NETWORK
TITLE = **** 7.2 - Submodules - Command **** Check Received
// Check Received Data
      AN    #SendAckCmd;  // Send AckCmd
      JC    SACK;
      L     #OldRecMsgNbr;  // MessageNumber (SeqNbr)
      OPN   #I_VDCommSendDB;
      T     %DBW8;
      L     #OldSubSystem;  // Subsystem
      T     %DBW6;
      L     1;  // MessageType
      T     %DBW4;
      L     10;  //LengthLength
      T     %DBW2;
      JU    PAPM;
SACK: NOP   0;

      AN    #SendNackCmd;  // Send NackCmd
      JC    SNAC;
      L     #OldRecMsgNbr;  // MessageNumber (SeqNbr)
      OPN   #I_VDCommSendDB;
      T     %DBW8;
      L     #OldSubSystem;  // Subsystem
      T     %DBW6;
      L     0;  // MessageType
      T     %DBW4;
      L     10;  //LengthLength
      T     %DBW2;
      JU    PAPM;
SNAC: NOP   0;

      A     #SendApplMsgCmd;  // Send Application Message
      AN    #SendActive;
      AN    #SendDone;
      JCN   PAPM;

// Number of bytes to copy***************************************************************************************************
//     L     #I_VDCommSendDBBuf   // SEND BUF        APa Fixa S7-1500
//     T     #SS_Out_Buf          // DB number to copy
//     OPN DB [ #SS_Out_Buf]      // APa Fixa S7-1500
//     OPN   #I_VDCommSendDBBuf

      L     #IO_VD.VDCommSendDBNr;
      L     0;
      ==I;
//     JCN   NSrS1
      OPN   #IO_VD.VDCommSendDB;
      L     DBNO;
      T     #OutBuf;
      OPN   #IO_VD.VDCommSendDB;
      LAR1  P##PointerSendBuf;
      L     %DBW2;  // Length
      T     LW [AR1, P#2.0];
      OPN   #IO_VD.VDCommSendDB;
      LAR1  P##PointerSend;
      L     %DBW2;
      T     LW [AR1, P#2.0];
      OPN   #IO_VD.VDCommSendDB;
      L     DBNO;
      T     #OutBuf;
//NSrS1: NOP 0

//      OPN   #I_VDCommSendBufStn2 APa Fixa S7-1500
//    L DBNO
//   L     #I_VDCommSendDBBuf
//    ==I
//    L DBNO
//     T     #SS_Out_Buf
//     JCN   NSrS2
//      OPN   #I_VDCommSendBufStn2
//    L     %DBW2                // Length
//    T     %LW22                // SEND BUF
//     T     %LW12                // SEND
//     L DBNO
//      T     #SS_Out_Buf
//NSrS2: NOP 0

//*****************************************************************************************************************************


// Pointer to the Receive DB (Pointer_SEND_Buf) APa Fixa S7-1500
// DB no DB no
//    L DBNO
//  T     #SS_Out_Buf
//   L     #I_VDCommSendDBBuf
      OPN   #IO_VD.VDCommSendDB;
      L     DBNO;
      T     #OutBuf;
      L     #OutBuf;
      LAR1  P##PointerSendBuf;
      L     #OutBuf;
      T     LW [AR1, P#4.0];
//      T     %LW24                // SEND BUF
      CALL  BLKMOV
      ( SRCBLK  := #PointerSendBuf,  // SEND Buffer
        RET_VAL := "NotUsedInt",
        DSTBLK  := #PointerSend  // SEND
      );  // Copy data from buffer DB to send DB

      L     #SendMsgNbr;
      L     1000;
      >=I;
      JCN   ZermMsgCnt;
      L     1;
      T     #SendMsgNbr;

ZermMsgCnt:OPN   #I_VDCommSendDB;
      L     #SendMsgNbr;
      A     #AD_TimeoutApplMsgMem;
      JC    noin;
      L     #SendMsgNbr;
      +     1;
noin: T     #SendMsgNbr;
      T     %DBW8;  // Messagenumber

      CLR;
      R     #AD_TimeoutApplMsgMem;

PAPM: OPN   #I_VDCommSendDB;
      L     %DBW2;
      T     #MsgLen;

      L     1;
      T     %DBB0;

      A     #NackIsLastSent;
      A     #SendAckCmd;
      JCN   ZeroMesag;
      L     0;
      T     %DBW4;
ZeroMesag:NOP   0;

      L     #SendMsgNbr;
      T     "NotUsedDInt";

NETWORK
TITLE = **** 7.2 - Submodules - Command **** Length to Send Pointers
// Length to Send Pointers / Check Received Data
      LAR1  P##PointerSend;
      L     #MsgLen;
      T     LW [AR1, P#2.0];


REGION Network 73: **** 7.2 - Submodules - Command **** Send Data VD
   // Send Data VD
   #_w1 := (#SendNackCmd OR #SendAckCmd OR #SendApplMsgCmd OR #SendKeepAliveCmd) AND NOT #HMIResetAndInit AND NOT #SendActive;
   IF "TRUE" THEN
       #TSendVD(REQ := #_w1,   // TSEND
                ID := #ConnectionSettings.ID,
                LEN := #MsgLen,
                DATA := #PointerSend,
                DONE => #TSEND.Done,
                BUSY => #TSEND.Busy,
                ERROR => #TSEND.Error,
                STATUS => #TSEND.Status);
   END_IF;
   IF #_w1 THEN #TSEND.Sending := TRUE; END_IF;
END_REGION

NETWORK
TITLE = **** 7.2 - Submodules - Command **** Send Data to VD
// Send data to VD (length is the length in the SEND_DB)
      L     #TSEND.Status;
      L     16#0000;
      ==I;
      =     #SendJobCompleted;  // Send job completed without error
      L     #TSEND.Status;
      L     16#7000;
      ==I;
      =     #SendInactive;  // No job processing active
      L     #TSEND.Status;
      L     16#7001;
      ==I;
      =     #SendStartOfProc;  // Start of job processing, data being sent
      L     #TSEND.Status;
      L     16#7002;
      ==I;
      =     #SendFollowOnCall;  // Follow-on call (REQ irrelevant ), job being processed



REGION Network 75: **** 7.2 - Submodules - Command **** Send Status
   // Send Status to memory
   IF #TSEND.Error THEN #TSEND.Status_Mem := #TSEND.Status; END_IF;
END_REGION

REGION Network 76: **** 7.2 - Submodules - Command **** Stop Send
   // Stop sending  Error,Done,Sending AND NOT Busy
   IF (#TSEND.Sending AND NOT #TSEND.Busy AND #AD_SendTimeOut) OR #TSEND.Error OR #TSEND.Done THEN
       #TSEND.Sending := FALSE;
   END_IF;
END_REGION

REGION Network 77: **** 7.2 - Submodules - Command **** Send Active
   // Send Active
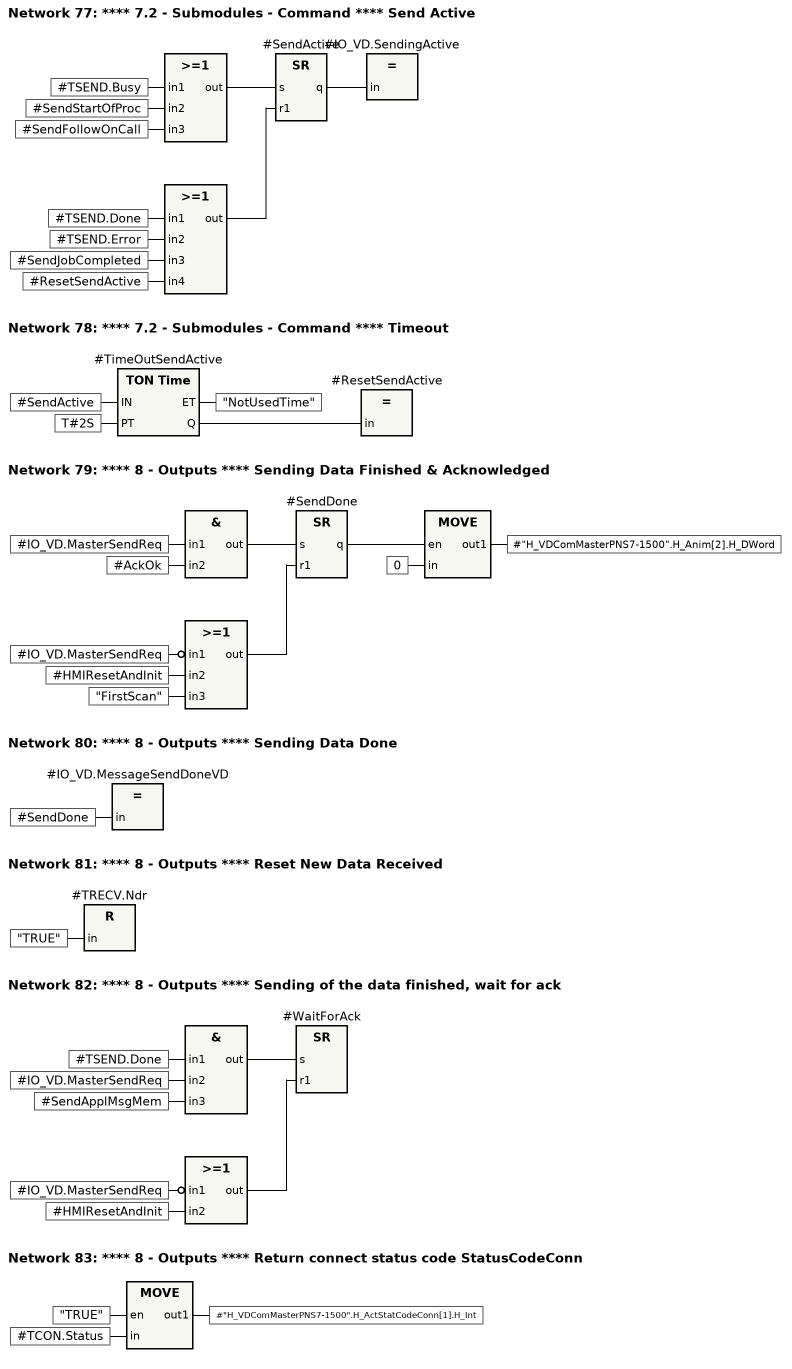
   IF #TSEND.Busy OR #SendStartOfProc OR #SendFollowOnCall THEN
       #SendActive := TRUE;   // SR flip-flop
   END_IF;
   IF #TSEND.Done OR #TSEND.Error OR #SendJobCompleted OR #ResetSendActive THEN #SendActive := FALSE; END_IF;
   #IO_VD.SendingActive := #SendActive;
END_REGION

REGION Network 78: **** 7.2 - Submodules - Command **** Timeout
   // Timeout
   #TimeOutSendActive(IN := #SendActive, PT := T#2S, ET => "NotUsedTime");   // TON
   #ResetSendActive := #TimeOutSendActive.Q;
END_REGION

REGION Network 79: **** 8 - Outputs **** Sending Data Finished & Acknowledged
   // Sending Data Finished & Acknowledged
   IF #IO_VD.MasterSendReq AND #AckOk THEN
       #SendDone := TRUE;   // SR flip-flop
   END_IF;
   IF NOT #IO_VD.MasterSendReq OR #HMIResetAndInit OR "FirstScan" THEN #SendDone := FALSE; END_IF;
   IF #SendDone THEN #"H_VDComMasterPNS7-1500".H_Anim[2].H_DWord := 0; END_IF;
END_REGION

REGION Network 80: **** 8 - Outputs **** Sending Data Done
   // Sending Data Done
   #IO_VD.MessageSendDoneVD := #SendDone;
END_REGION

REGION Network 81: **** 8 - Outputs **** Reset New Data Received
   // Reset "New data received" bit. All processing shall be done before this step.
   IF "TRUE" THEN #TRECV.Ndr := FALSE; END_IF;
END_REGION

REGION Network 82: **** 8 - Outputs **** Sending of the data finished, wait for ack
   // Sending of the data finished, wait for ack
   IF #TSEND.Done AND #IO_VD.MasterSendReq AND #SendApplMsgMem THEN
       #WaitForAck := TRUE;   // SR flip-flop
   END_IF;
   IF NOT #IO_VD.MasterSendReq OR #HMIResetAndInit THEN #WaitForAck := FALSE; END_IF;
END_REGION

REGION Network 83: **** 8 - Outputs **** Return connect status code StatusCodeConn
   // Return connect status code H_StatusCodeConn
   IF "TRUE" THEN #"H_VDComMasterPNS7-1500".H_ActStatCodeConn[1].H_Int := #TCON.Status; END_IF;
END_REGION

REGION Network 84: **** 8 - Outputs **** Return receive status code StatusCodeDisconn
   // Return receive status code H_StatusCodeDisconn
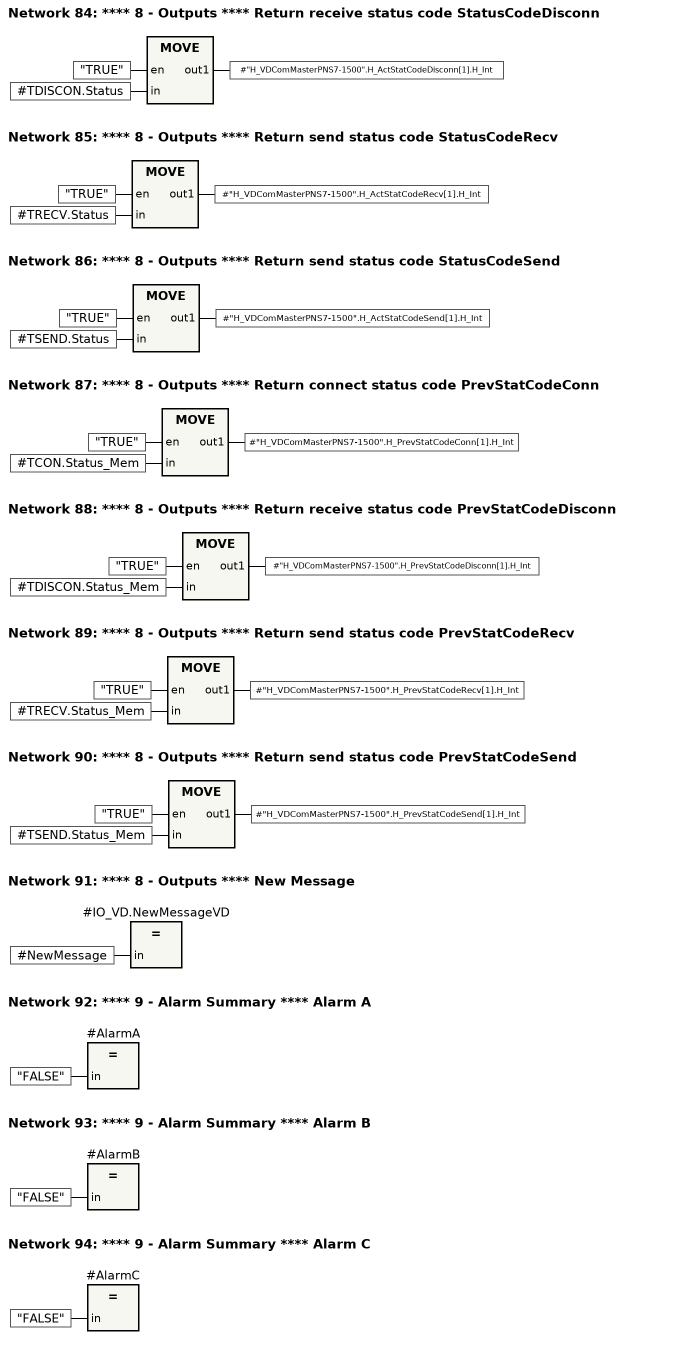
   IF "TRUE" THEN #"H_VDComMasterPNS7-1500".H_ActStatCodeDisconn[1].H_Int := #TDISCON.Status; END_IF;
END_REGION

REGION Network 85: **** 8 - Outputs **** Return send status code StatusCodeRecv
   // Return send status code H_StatusCodeRecv
   IF "TRUE" THEN #"H_VDComMasterPNS7-1500".H_ActStatCodeRecv[1].H_Int := #TRECV.Status; END_IF;
END_REGION

REGION Network 86: **** 8 - Outputs **** Return send status code StatusCodeSend
   // Return send status code H_StatusCodeSend
   IF "TRUE" THEN #"H_VDComMasterPNS7-1500".H_ActStatCodeSend[1].H_Int := #TSEND.Status; END_IF;
END_REGION

REGION Network 87: **** 8 - Outputs **** Return connect status code PrevStatCodeConn
   // Return connect status code H_PrevStatCodeConn
   IF "TRUE" THEN #"H_VDComMasterPNS7-1500".H_PrevStatCodeConn[1].H_Int := #TCON.Status_Mem; END_IF;
END_REGION

REGION Network 88: **** 8 - Outputs **** Return receive status code PrevStatCodeDisconn
   // Return receive status code H_PrevStatCodeDisconn
   IF "TRUE" THEN #"H_VDComMasterPNS7-1500".H_PrevStatCodeDisconn[1].H_Int := #TDISCON.Status_Mem; END_IF;
END_REGION

REGION Network 89: **** 8 - Outputs **** Return send status code PrevStatCodeRecv
   // Return send status code H_PrevStatCodeRecv
   IF "TRUE" THEN #"H_VDComMasterPNS7-1500".H_PrevStatCodeRecv[1].H_Int := #TRECV.Status_Mem; END_IF;
END_REGION

REGION Network 90: **** 8 - Outputs **** Return send status code PrevStatCodeSend
   // Return send status code H_PrevStatCodeSend
   IF "TRUE" THEN #"H_VDComMasterPNS7-1500".H_PrevStatCodeSend[1].H_Int := #TSEND.Status_Mem; END_IF;
END_REGION

REGION Network 91: **** 8 - Outputs **** New Message
   // New Message
   #IO_VD.NewMessageVD := #NewMessage;
END_REGION

REGION Network 92: **** 9 - Alarm Summary **** Alarm A
   // Alarm A
   #AlarmA := "FALSE";
END_REGION

REGION Network 93: **** 9 - Alarm Summary **** Alarm B
   // Alarm B
   #AlarmB := "FALSE";
END_REGION

REGION Network 94: **** 9 - Alarm Summary **** Alarm C
   // Alarm C
   #AlarmC := "FALSE";
END_REGION

REGION Network 95: **** 9 - Alarm Summary **** Alarm D
   // Alarm D
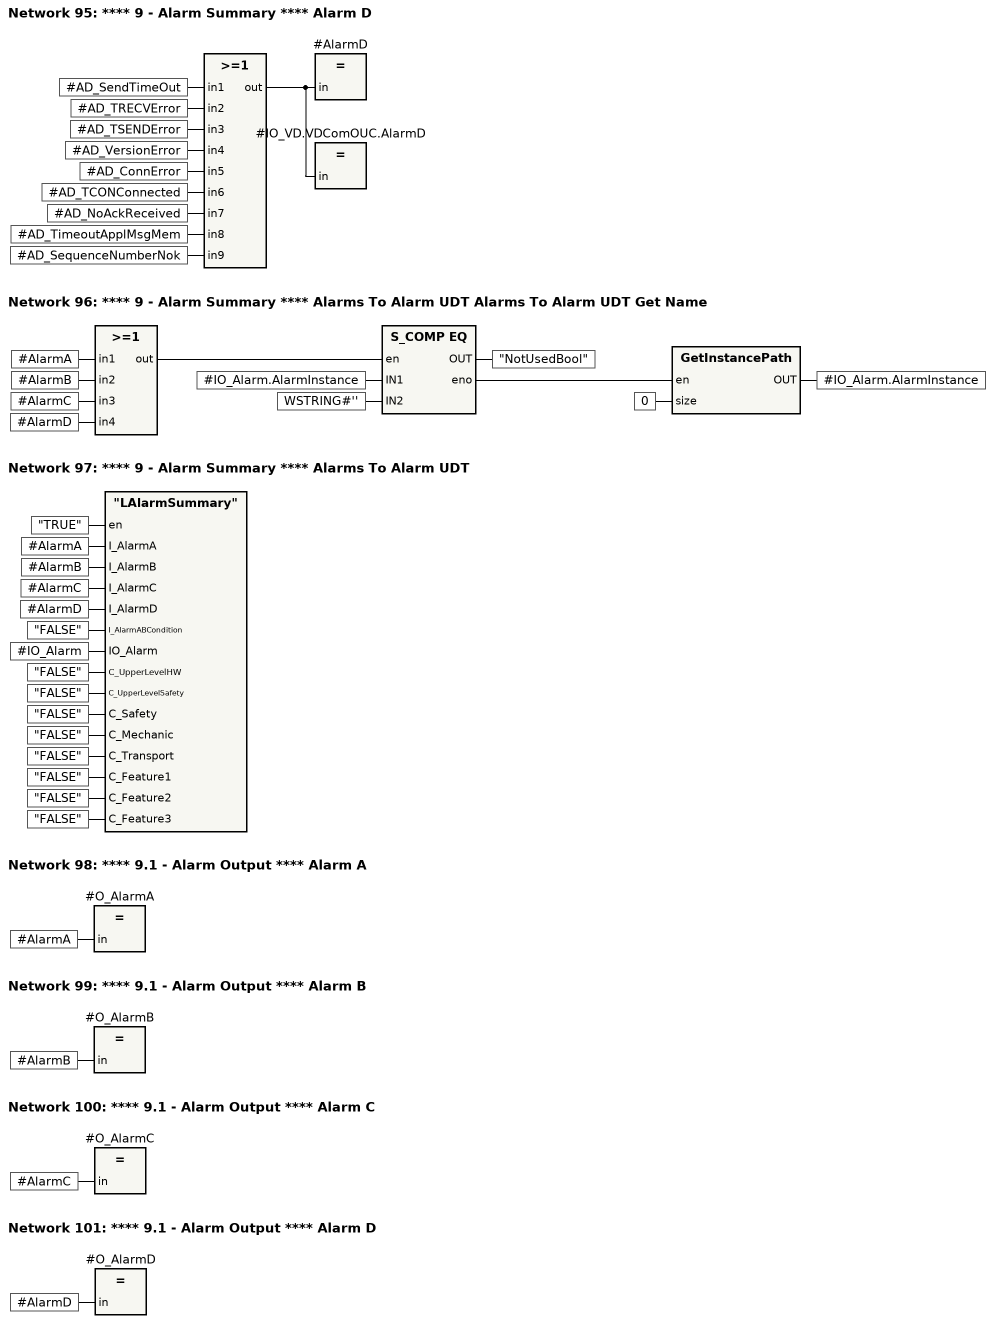
   #AlarmD := #AD_SendTimeOut OR #AD_TRECVError OR #AD_TSENDError OR #AD_VersionError OR #AD_ConnError OR #AD_TCONConnected OR #AD_NoAckReceived OR #AD_TimeoutApplMsgMem OR #AD_SequenceNumberNok;
   #IO_VD.VDComOUC.AlarmD := #AlarmD;
END_REGION

REGION Network 96: **** 9 - Alarm Summary **** Alarms To Alarm UDT Alarms To Alarm UDT Get Name
   // Alarm / Alarm D
   S_COMP(EN := #AlarmA OR #AlarmB OR #AlarmC OR #AlarmD,
          IN1 := #IO_Alarm.AlarmInstance,
          IN2 := WSTRING#'',
          OUT => "NotUsedBool",
          ENO => #_w1);
   IF #_w1 THEN GetInstancePath(size := 0, OUT => #IO_Alarm.AlarmInstance); END_IF;
END_REGION

REGION Network 97: **** 9 - Alarm Summary **** Alarms To Alarm UDT
   // Alarm / Alarm D
   IF "TRUE" THEN
       "LAlarmSummary"(I_AlarmA := #AlarmA,
                       I_AlarmB := #AlarmB,
                       I_AlarmC := #AlarmC,
                       I_AlarmD := #AlarmD,
                       I_AlarmABCondition := "FALSE",
                       IO_Alarm := #IO_Alarm,
                       C_UpperLevelHW := "FALSE",
                       C_UpperLevelSafety := "FALSE",
                       C_Safety := "FALSE",
                       C_Mechanic := "FALSE",
                       C_Transport := "FALSE",
                       C_Feature1 := "FALSE",
                       C_Feature2 := "FALSE",
                       C_Feature3 := "FALSE");
   END_IF;
END_REGION

REGION Network 98: **** 9.1 - Alarm Output **** Alarm A
   // Alarm A
   #O_AlarmA := #AlarmA;
END_REGION

REGION Network 99: **** 9.1 - Alarm Output **** Alarm B
   // Alarm B
   #O_AlarmB := #AlarmB;
END_REGION

REGION Network 100: **** 9.1 - Alarm Output **** Alarm C
   // Alarm C
   #O_AlarmC := #AlarmC;
END_REGION

REGION Network 101: **** 9.1 - Alarm Output **** Alarm D
   // Alarm D
   #O_AlarmD := #AlarmD;
END_REGION

REGION Network 102: **** 9.2 - Alarm DWord**** Alarm To DWord
   // Alarm To Word
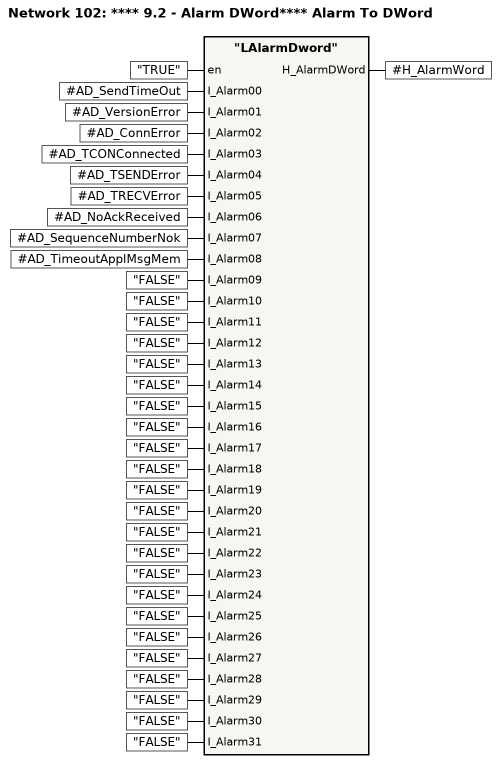
   IF "TRUE" THEN
       "LAlarmDword"(I_Alarm00 := #AD_SendTimeOut,
                     I_Alarm01 := #AD_VersionError,
                     I_Alarm02 := #AD_ConnError,
                     I_Alarm03 := #AD_TCONConnected,
                     I_Alarm04 := #AD_TSENDError,
                     I_Alarm05 := #AD_TRECVError,
                     I_Alarm06 := #AD_NoAckReceived,
                     I_Alarm07 := #AD_SequenceNumberNok,
                     I_Alarm08 := #AD_TimeoutApplMsgMem,
                     I_Alarm09 := "FALSE",
                     I_Alarm10 := "FALSE",
                     I_Alarm11 := "FALSE",
                     I_Alarm12 := "FALSE",
                     I_Alarm13 := "FALSE",
                     I_Alarm14 := "FALSE",
                     I_Alarm15 := "FALSE",
                     I_Alarm16 := "FALSE",
                     I_Alarm17 := "FALSE",
                     I_Alarm18 := "FALSE",
                     I_Alarm19 := "FALSE",
                     I_Alarm20 := "FALSE",
                     I_Alarm21 := "FALSE",
                     I_Alarm22 := "FALSE",
                     I_Alarm23 := "FALSE",
                     I_Alarm24 := "FALSE",
                     I_Alarm25 := "FALSE",
                     I_Alarm26 := "FALSE",
                     I_Alarm27 := "FALSE",
                     I_Alarm28 := "FALSE",
                     I_Alarm29 := "FALSE",
                     I_Alarm30 := "FALSE",
                     I_Alarm31 := "FALSE",
                     H_AlarmDWord => #H_AlarmWord);
   END_IF;
END_REGION
END_FUNCTION_BLOCK

FUNCTION_BLOCK "LPNIODiagIPS7-1500"   // FB2211, SCL
{ S7_Optimized_Access := 'TRUE' }
VERSION : 0.1
// stored: AutoNumber false, IsIECCheckEnabled false, IsRetainMemResEnabled false, MemoryReserve 100, SetENOAutomatically False, UDAEnableTagReadback false
   VAR_INPUT
      I_StartFillList { ExternalAccessible := 'False'; ExternalVisible := 'False'; ExternalWritable := 'False'} : Bool;
      I_LastDeviceNumber { ExternalAccessible := 'False'; ExternalVisible := 'False'; ExternalWritable := 'False'} : Int;   // Last Device of ProfiNet System
   END_VAR
   VAR_OUTPUT
      O_Done { ExternalAccessible := 'False'; ExternalVisible := 'False'; ExternalWritable := 'False'} : Bool;
      O_IPAddress { ExternalAccessible := 'False'; ExternalVisible := 'False'; ExternalWritable := 'False'} : Array[0..255] of String[15];
   END_VAR
   VAR_IN_OUT
      IO_DeviceExist : Array[0..255] of Bool;   // IO devices exist
      IO_HWIdentifier : Array[0..255] of UInt;   // HW Device
      IO_GetStationIP : Array[0..255] of IF_CONF_v4;   // Read out Station Information
   END_VAR
   VAR
      Index { ExternalAccessible := 'False'; ExternalVisible := 'False'; ExternalWritable := 'False'} : Int;
      LastDeviceNumber { ExternalAccessible := 'False'; ExternalVisible := 'False'; ExternalWritable := 'False'} : Int;   // Last Device of ProfiNet System
      Done { ExternalAccessible := 'False'; ExternalVisible := 'False'; ExternalWritable := 'False'} : Bool;
      DoneDelay { ExternalAccessible := 'False'; ExternalVisible := 'False'; ExternalWritable := 'False'} : Bool;
      ReturnGetStationInfoBusy_IP { ExternalAccessible := 'False'; ExternalVisible := 'False'; ExternalWritable := 'False'} : Bool;   // Temp
      ReturnGetStationInfoDone_IP { ExternalAccessible := 'False'; ExternalVisible := 'False'; ExternalWritable := 'False'} : Bool;   // Temp
      ReturnGetStationInfoError_IP { ExternalAccessible := 'False'; ExternalVisible := 'False'; ExternalWritable := 'False'} : Bool;   // Temp
      ReturnGetStationInfoStatus_IP { ExternalAccessible := 'False'; ExternalVisible := 'False'; ExternalWritable := 'False'} : Word;   // Temp
      IPAddress_ADDR1 { ExternalAccessible := 'False'; ExternalVisible := 'False'; ExternalWritable := 'False'} : String;
      IPAddress_ADDR2 { ExternalAccessible := 'False'; ExternalVisible := 'False'; ExternalWritable := 'False'} : String;
      IPAddress_ADDR3 { ExternalAccessible := 'False'; ExternalVisible := 'False'; ExternalWritable := 'False'} : String;
      IPAddress_ADDR4 { ExternalAccessible := 'False'; ExternalVisible := 'False'; ExternalWritable := 'False'} : String;
      IPAddress { ExternalAccessible := 'False'; ExternalVisible := 'False'; ExternalWritable := 'False'} : String[15];
      GetStationInfo_IP { ExternalAccessible := 'False'; ExternalVisible := 'False'; ExternalWritable := 'False'; S7_SetPoint := 'True'} : GetStationInfo;   // Get Station
      TimerDone { ExternalAccessible := 'False'; ExternalVisible := 'False'; ExternalWritable := 'False'; S7_SetPoint := 'True'} : TON_TIME;
      EdgeStartFillList { ExternalAccessible := 'False'; ExternalVisible := 'False'; ExternalWritable := 'False'; S7_SetPoint := 'True'} : R_TRIG;
   END_VAR
BEGIN
   #EdgeStartFillList(CLK:=#I_StartFillList);

   IF #EdgeStartFillList.Q THEN
       #Done := False;
       #Index := 0;
   END_IF;

   #LastDeviceNumber := #I_LastDeviceNumber;
   IF #I_LastDeviceNumber < 1 THEN
       #LastDeviceNumber := 1;
   END_IF;
   IF #I_LastDeviceNumber > 254 THEN
       #LastDeviceNumber := 254;
   END_IF;

   #TimerDone(IN := #Done,
              PT := T#500ms,
              Q => #DoneDelay);

   IF (#I_StartFillList & NOT #Done) THEN
       #Index := #Index + 1;
       WHILE (#IO_DeviceExist[#Index] & NOT #ReturnGetStationInfoDone_IP) DO
               #GetStationInfo_IP(REQ := #IO_DeviceExist[#Index] & NOT #ReturnGetStationInfoBusy_IP,
                      LADDR := #IO_HWIdentifier[#Index],
                      MODE := 1,
                      DONE => #ReturnGetStationInfoDone_IP,
                      BUSY => #ReturnGetStationInfoBusy_IP,
                      ERROR => #ReturnGetStationInfoError_IP,
                      STATUS => #ReturnGetStationInfoStatus_IP,
                      DATA := #IO_GetStationIP[#Index]);
        END_WHILE;
        #ReturnGetStationInfoDone_IP := False;

       VAL_STRG(IN := BYTE_TO_USINT(#IO_GetStationIP[#Index].InterfaceAddress.ADDR[1]),
                SIZE := 3,
                PREC := 0,
                FORMAT := 16#0000,
                P := 1,
                OUT => #IPAddress_ADDR1);
       VAL_STRG(IN := BYTE_TO_USINT(#IO_GetStationIP[#Index].InterfaceAddress.ADDR[2]),
                SIZE := 3,
                PREC := 0,
                FORMAT := 16#0000,
                P := 1,
                OUT => #IPAddress_ADDR2);
       VAL_STRG(IN := BYTE_TO_USINT(#IO_GetStationIP[#Index].InterfaceAddress.ADDR[3]),
                SIZE := 3,
                PREC := 0,
                FORMAT := 16#0000,
                P := 1,
                OUT => #IPAddress_ADDR3);
       VAL_STRG(IN := BYTE_TO_USINT(#IO_GetStationIP[#Index].InterfaceAddress.ADDR[4]),
                SIZE := 3,
                PREC := 0,
                FORMAT := 16#0000,
                P := 1,
                OUT => #IPAddress_ADDR4);

       #IPAddress := CONCAT_STRING(IN1 := #IPAddress_ADDR1, IN2 :='.');
       #IPAddress := CONCAT_STRING(IN1 := #IPAddress, IN2 := #IPAddress_ADDR2);
       #IPAddress := CONCAT_STRING(IN1 := #IPAddress, IN2 := '.');
       #IPAddress := CONCAT_STRING(IN1 := #IPAddress, IN2 := #IPAddress_ADDR3);
       #IPAddress := CONCAT_STRING(IN1 := #IPAddress, IN2 := '.');
       #IPAddress := CONCAT_STRING(IN1 := #IPAddress, IN2 := #IPAddress_ADDR4);
       #O_IPAddress[#Index] := #IPAddress;
       IF #Index = #LastDeviceNumber THEN
           #Done := True;
       END_IF;
   END_IF;

   #O_Done := #DoneDelay;
END_FUNCTION_BLOCK

FUNCTION_BLOCK "LPNIODiagMACS7-1500"   // FB2212, SCL
{ S7_Optimized_Access := 'TRUE' }
VERSION : 0.1
// stored: AutoNumber false, IsIECCheckEnabled false, IsRetainMemResEnabled false, MemoryReserve 100, SetENOAutomatically False, UDAEnableTagReadback false
   VAR_INPUT
      I_StartFillList { ExternalAccessible := 'False'; ExternalVisible := 'False'; ExternalWritable := 'False'} : Bool;
      I_LastDeviceNumber { ExternalAccessible := 'False'; ExternalVisible := 'False'; ExternalWritable := 'False'} : Int;   // Last Device of ProfiNet System
   END_VAR
   VAR_OUTPUT
      O_Done { ExternalAccessible := 'False'; ExternalVisible := 'False'; ExternalWritable := 'False'} : Bool;
      O_MACAddress { ExternalAccessible := 'False'; ExternalVisible := 'False'; ExternalWritable := 'False'} : Array[0..255] of String[18];
   END_VAR
   VAR_IN_OUT
      IO_DeviceExist : Array[0..255] of Bool;   // IO devices exist
      IO_HWIdentifier : Array[0..255] of UInt;   // HW Device
      IO_GetStationMAC : Array[0..255] of IF_CONF_MAC;   // Read out Station Information
   END_VAR
   VAR
      Index { ExternalAccessible := 'False'; ExternalVisible := 'False'; ExternalWritable := 'False'} : Int;
      LastDeviceNumber { ExternalAccessible := 'False'; ExternalVisible := 'False'; ExternalWritable := 'False'} : Int;   // Last Device of ProfiNet System
      Done { ExternalAccessible := 'False'; ExternalVisible := 'False'; ExternalWritable := 'False'} : Bool;
      DoneDelay { ExternalAccessible := 'False'; ExternalVisible := 'False'; ExternalWritable := 'False'} : Bool;
      ReturnGetStationInfoBusy_MAC { ExternalAccessible := 'False'; ExternalVisible := 'False'; ExternalWritable := 'False'} : Bool;   // Temp
      ReturnGetStationInfoDone_MAC { ExternalAccessible := 'False'; ExternalVisible := 'False'; ExternalWritable := 'False'} : Bool;   // Temp
      ReturnGetStationInfoError_MAC { ExternalAccessible := 'False'; ExternalVisible := 'False'; ExternalWritable := 'False'} : Bool;   // Temp
      ReturnGetStationInfoStatus_MAC { ExternalAccessible := 'False'; ExternalVisible := 'False'; ExternalWritable := 'False'} : Word;   // Temp
      MACAddress_ADDR1 { ExternalAccessible := 'False'; ExternalVisible := 'False'; ExternalWritable := 'False'} : String[2];
      MACAddress_ADDR2 { ExternalAccessible := 'False'; ExternalVisible := 'False'; ExternalWritable := 'False'} : String[2];
      MACAddress_ADDR3 { ExternalAccessible := 'False'; ExternalVisible := 'False'; ExternalWritable := 'False'} : String[2];
      MACAddress_ADDR4 { ExternalAccessible := 'False'; ExternalVisible := 'False'; ExternalWritable := 'False'} : String[2];
      MACAddress_ADDR5 { ExternalAccessible := 'False'; ExternalVisible := 'False'; ExternalWritable := 'False'} : String[2];
      MACAddress_ADDR6 { ExternalAccessible := 'False'; ExternalVisible := 'False'; ExternalWritable := 'False'} : String[2];
      MACAddress { ExternalAccessible := 'False'; ExternalVisible := 'False'; ExternalWritable := 'False'} : String[18];
      RetVal { ExternalAccessible := 'False'; ExternalVisible := 'False'; ExternalWritable := 'False'} : Word;
      GetStationInfo_MAC { ExternalAccessible := 'False'; ExternalVisible := 'False'; ExternalWritable := 'False'; S7_SetPoint := 'True'} : GetStationInfo;
      TimerDone { ExternalAccessible := 'False'; ExternalVisible := 'False'; ExternalWritable := 'False'; S7_SetPoint := 'True'} : TON_TIME;
      EdgeStartFillList { ExternalAccessible := 'False'; ExternalVisible := 'False'; ExternalWritable := 'False'; S7_SetPoint := 'True'} : R_TRIG;
   END_VAR
BEGIN
   #EdgeStartFillList(CLK := #I_StartFillList);

   IF #EdgeStartFillList.Q THEN
       #Done := False;
       #Index := 0;
   END_IF;

   #LastDeviceNumber := #I_LastDeviceNumber;
   IF #I_LastDeviceNumber < 1 THEN
       #LastDeviceNumber := 1;
   END_IF;
   IF #I_LastDeviceNumber > 254 THEN
       #LastDeviceNumber := 254;
   END_IF;

   #TimerDone(IN := #Done,
              PT := T#500ms,
              Q => #DoneDelay);

   IF (#I_StartFillList & NOT #Done) THEN
       #Index := #Index + 1;
       WHILE (#IO_DeviceExist[#Index] & NOT #ReturnGetStationInfoDone_MAC) DO
           #GetStationInfo_MAC(REQ := #IO_DeviceExist[#Index] & NOT #ReturnGetStationInfoBusy_MAC,
               LADDR := #IO_HWIdentifier[#Index],
               MODE := 2,
               DONE => #ReturnGetStationInfoDone_MAC,
               BUSY => #ReturnGetStationInfoBusy_MAC,
               ERROR => #ReturnGetStationInfoError_MAC,
               STATUS => #ReturnGetStationInfoStatus_MAC,
               DATA := #IO_GetStationMAC[#Index]);
       END_WHILE;
       #ReturnGetStationInfoDone_MAC := False;

       #RetVal := HTA(IN := #IO_GetStationMAC[#Index].Mac[1], N := 2, OUT => #MACAddress_ADDR1);
       #RetVal := HTA(IN := #IO_GetStationMAC[#Index].Mac[2], N := 2, OUT => #MACAddress_ADDR2);
       #RetVal := HTA(IN := #IO_GetStationMAC[#Index].Mac[3], N := 2, OUT => #MACAddress_ADDR3);
       #RetVal := HTA(IN := #IO_GetStationMAC[#Index].Mac[4], N := 2, OUT => #MACAddress_ADDR4);
       #RetVal := HTA(IN := #IO_GetStationMAC[#Index].Mac[5], N := 2, OUT => #MACAddress_ADDR5);
       #RetVal := HTA(IN := #IO_GetStationMAC[#Index].Mac[6], N := 2, OUT => #MACAddress_ADDR6);

       #MACAddress := CONCAT_STRING(IN1 := #MACAddress_ADDR1, IN2 := '.');
       #MACAddress := CONCAT_STRING(IN1 := #MACAddress, IN2 := #MACAddress_ADDR2);
       #MACAddress := CONCAT_STRING(IN1 := #MACAddress, IN2 := '.');
       #MACAddress := CONCAT_STRING(IN1 := #MACAddress, IN2 := #MACAddress_ADDR3);
       #MACAddress := CONCAT_STRING(IN1 := #MACAddress, IN2 := '.');
       #MACAddress := CONCAT_STRING(IN1 := #MACAddress, IN2 := #MACAddress_ADDR4);
       #MACAddress := CONCAT_STRING(IN1 := #MACAddress, IN2 := '.');
       #MACAddress := CONCAT_STRING(IN1 := #MACAddress, IN2 := #MACAddress_ADDR5);
       #MACAddress := CONCAT_STRING(IN1 := #MACAddress, IN2 := '.');
       #MACAddress := CONCAT_STRING(IN1 := #MACAddress, IN2 := #MACAddress_ADDR6);
       #O_MACAddress[#Index] := #MACAddress;
       IF #Index = #LastDeviceNumber THEN
           #Done := True;
       END_IF;
   END_IF;

   #O_Done := #DoneDelay;
END_FUNCTION_BLOCK

FUNCTION_BLOCK "LPNIODiagNameS7-1500"   // FB2213, SCL
{ S7_Optimized_Access := 'TRUE' }
VERSION : 0.1
// stored: AutoNumber false, IsIECCheckEnabled false, IsRetainMemResEnabled false, MemoryReserve 100, SetENOAutomatically False, UDAEnableTagReadback false
   VAR_INPUT
      I_StartFillList { ExternalAccessible := 'False'; ExternalVisible := 'False'; ExternalWritable := 'False'} : Bool;
      I_LastDeviceNumber { ExternalAccessible := 'False'; ExternalVisible := 'False'; ExternalWritable := 'False'} : Int;   // Last Device of ProfiNet System
      I_HWIOSYSTEM { ExternalAccessible := 'False'; ExternalVisible := 'False'; ExternalWritable := 'False'} : HW_IOSYSTEM;   // HW ID ProfiNet System
   END_VAR
   VAR_OUTPUT
      O_Done { ExternalAccessible := 'False'; ExternalVisible := 'False'; ExternalWritable := 'False'} : Bool;
      O_Name { ExternalAccessible := 'False'; ExternalVisible := 'False'; ExternalWritable := 'False'} : Array[0..255] of String[25];
   END_VAR
   VAR_IN_OUT
      IO_DeviceExist : Array[0..255] of Bool;   // IO devices exist
      IO_GetStationName : Array[0..255] of String;   // Profinet Name
   END_VAR
   VAR
      Index { ExternalAccessible := 'False'; ExternalVisible := 'False'; ExternalWritable := 'False'} : Int;
      LastDeviceNumber { ExternalAccessible := 'False'; ExternalVisible := 'False'; ExternalWritable := 'False'} : Int;   // Last Device of ProfiNet System
      Done { ExternalAccessible := 'False'; ExternalVisible := 'False'; ExternalWritable := 'False'} : Bool;
      DoneDelay { ExternalAccessible := 'False'; ExternalVisible := 'False'; ExternalWritable := 'False'} : Bool;
      ReturnGetNameBusy { ExternalAccessible := 'False'; ExternalVisible := 'False'; ExternalWritable := 'False'} : Bool;   // Temp
      ReturnGetNameDone { ExternalAccessible := 'False'; ExternalVisible := 'False'; ExternalWritable := 'False'} : Bool;   // Temp
      ReturnGetNameError { ExternalAccessible := 'False'; ExternalVisible := 'False'; ExternalWritable := 'False'} : Bool;   // Temp
      ReturnGetNameLen { ExternalAccessible := 'False'; ExternalVisible := 'False'; ExternalWritable := 'False'} : DInt;   // Temp
      ReturnGetNameStatus { ExternalAccessible := 'False'; ExternalVisible := 'False'; ExternalWritable := 'False'} : Word;   // Temp
      GetNameInstance { ExternalAccessible := 'False'; ExternalVisible := 'False'; ExternalWritable := 'False'; S7_SetPoint := 'True'} : Get_Name;   // Get Name of Devices
      TimerDone { ExternalAccessible := 'False'; ExternalVisible := 'False'; ExternalWritable := 'False'; S7_SetPoint := 'True'} : TON_TIME;
      EdgeStartFillList { ExternalAccessible := 'False'; ExternalVisible := 'False'; ExternalWritable := 'False'; S7_SetPoint := 'True'} : R_TRIG;
   END_VAR
BEGIN
   #EdgeStartFillList(CLK := #I_StartFillList);

   IF #EdgeStartFillList.Q THEN
       #Done := False;
       #Index := 0;
   END_IF;

   #LastDeviceNumber := #I_LastDeviceNumber;
   IF #I_LastDeviceNumber < 1 THEN
       #LastDeviceNumber := 1;
   END_IF;
   IF #I_LastDeviceNumber > 254 THEN
       #LastDeviceNumber := 254;
   END_IF;


   #TimerDone(IN := #Done,
              PT := T#500ms,
              Q => #DoneDelay);

   IF (#I_StartFillList & NOT #Done) THEN
       #Index := #Index + 1;
       IF #IO_DeviceExist[#Index] THEN
           WHILE (#IO_DeviceExist[#Index] & NOT #ReturnGetNameDone) DO
               #GetNameInstance(LADDR := #I_HWIOSYSTEM,
                    STATION_NR := INT_TO_UINT(#Index),
                    DONE => #ReturnGetNameDone,
                    BUSY => #ReturnGetNameBusy,
                    ERROR => #ReturnGetNameError,
                    LEN => #ReturnGetNameLen,
                    STATUS => #ReturnGetNameStatus,
                    DATA := #IO_GetStationName[#Index]);
           END_WHILE;
           #ReturnGetNameDone := False;

           #O_Name[#Index] := #IO_GetStationName[#Index];
       END_IF;
       IF #Index = #LastDeviceNumber THEN
           #Done := True;
       END_IF;
   END_IF;

   #O_Done := #DoneDelay;
END_FUNCTION_BLOCK

FUNCTION_BLOCK "LPNIODiagHMIS7-1500"   // FB2214, FBD
TITLE = LPNIODiagHMIS7-1500
{ S7_Optimized_Access := 'FALSE' }
VERSION : 0.1
// stored: AutoNumber false, IsIECCheckEnabled false, SetENOAutomatically False, UDAEnableTagReadback false
   VAR_INPUT
      I_DeviceNumber { ExternalAccessible := 'False'; ExternalVisible := 'False'; ExternalWritable := 'False'} : Int;   // Device number in the hardware config
      I_Name { ExternalAccessible := 'False'; ExternalVisible := 'False'; ExternalWritable := 'False'} : String[25];   // Name device from list
      I_IPAddress { ExternalAccessible := 'False'; ExternalVisible := 'False'; ExternalWritable := 'False'} : String[15];   // IP address device from list
      I_MACAddress { ExternalAccessible := 'False'; ExternalVisible := 'False'; ExternalWritable := 'False'} : String[18];   // MAC address device from list
      I_AlarmClass { ExternalAccessible := 'False'; ExternalVisible := 'False'; ExternalWritable := 'False'} : Char;   // Alarm class -> A - B - C - D or E
      I_EnableAlarm { ExternalAccessible := 'False'; ExternalVisible := 'False'; ExternalWritable := 'False'} : Bool := TRUE;   // Enable alarm from upper level
      I_EnableButtons { ExternalAccessible := 'False'; ExternalVisible := 'False'; ExternalWritable := 'False'} : Bool;   // Enable to use the buttons in the pop-up -> "Activate" and "Deactivate"
   END_VAR
   VAR_OUTPUT
      O_Alarm { ExternalAccessible := 'False'; ExternalVisible := 'False'; ExternalWritable := 'False'} : Bool;   // Alarm A
      O_AC_Faulty { ExternalAccessible := 'False'; ExternalVisible := 'False'; ExternalWritable := 'False'} : Bool;   // Device is in faulty
      O_AD_Disabled { ExternalAccessible := 'False'; ExternalVisible := 'False'; ExternalWritable := 'False'} : Bool;   // Device is disabled
      O_AlarmABcondition { ExternalAccessible := 'False'; ExternalVisible := 'False'; ExternalWritable := 'False'} : Bool;   // Alarm AB condition
      H_IAnim { ExternalAccessible := 'False'; ExternalVisible := 'False'; ExternalWritable := 'False'} : Word;   // HMI Animation color of the icon
      H_IAnim2 { ExternalAccessible := 'False'; ExternalVisible := 'False'; ExternalWritable := 'False'} : Int;   // HMI Animation
   END_VAR
   VAR_IN_OUT
      IO_PNIODIAG_Global : "H_PNIODiagS7-1500";
   END_VAR
   VAR DB_SPECIFIC
      H_In : Struct   // HMI
         HMICmd : Word;   // Commands from HMI
         Mode : Int;   // Mode
      END_STRUCT;
      H_Out : Struct   // HMI
         Anim : Word;   // HMI Animation Word
         DeviceNumber : Int;   // HMI Device number (node)
         "Name" : String[25];   // HMI Profinet name
         IPAddress : String[15];   // HMI IP Address
         MACAddress : String[18];   // HMI MAC Address
         DBnr : Int;   // HMI Animation DB number
      END_STRUCT;
      HMICmdActivated { ExternalAccessible := 'False'; ExternalVisible := 'False'; ExternalWritable := 'False'} : Bool;   // HMI Cmd
      HMICmdDeactivated { ExternalAccessible := 'False'; ExternalVisible := 'False'; ExternalWritable := 'False'} : Bool;   // HMI Cmd
      Alarm { ExternalAccessible := 'False'; ExternalVisible := 'False'; ExternalWritable := 'False'} : Bool;   // Alarm
      AlarmClass_A { ExternalAccessible := 'False'; ExternalVisible := 'False'; ExternalWritable := 'False'} : Bool;   // The alarm is from alarm class A
      AlarmClass_B { ExternalAccessible := 'False'; ExternalVisible := 'False'; ExternalWritable := 'False'} : Bool;   // The alarm is from alarm class B
      AlarmClass_C { ExternalAccessible := 'False'; ExternalVisible := 'False'; ExternalWritable := 'False'} : Bool;   // The alarm is from alarm class C
      AlarmClass_D { ExternalAccessible := 'False'; ExternalVisible := 'False'; ExternalWritable := 'False'} : Bool;   // The alarm is from alarm class D
      AlarmClass_E { ExternalAccessible := 'False'; ExternalVisible := 'False'; ExternalWritable := 'False'} : Bool;   // The alarm is from alarm class E
      AlarmCond { ExternalAccessible := 'False'; ExternalVisible := 'False'; ExternalWritable := 'False'} : Bool;   // Alarm condition
      DBnr { ExternalAccessible := 'False'; ExternalVisible := 'False'; ExternalWritable := 'False'} : Int;   // HMI DB number
      DeviceExist { ExternalAccessible := 'False'; ExternalVisible := 'False'; ExternalWritable := 'False'} : Bool;   // Device exist
      DeviceDisabled { ExternalAccessible := 'False'; ExternalVisible := 'False'; ExternalWritable := 'False'} : Bool;   // Device is disabled
      DeviceFaulty { ExternalAccessible := 'False'; ExternalVisible := 'False'; ExternalWritable := 'False'} : Bool;   // Device is in faulty
      DeviceServiceReq { ExternalAccessible := 'False'; ExternalVisible := 'False'; ExternalWritable := 'False'} : Bool;   // Device has a service request
      EnableBtnActivate { ExternalAccessible := 'False'; ExternalVisible := 'False'; ExternalWritable := 'False'} : Bool;   // Enable button in pop-up
      EnableBtnDeactivate { ExternalAccessible := 'False'; ExternalVisible := 'False'; ExternalWritable := 'False'} : Bool;   // Enable button in pop-up
      TimerDeviceDisabled { ExternalAccessible := 'False'; ExternalVisible := 'False'; ExternalWritable := 'False'; S7_SetPoint := 'True'} : TOF_TIME;   // Timer
      TimerActivateDeactivateBusy { ExternalAccessible := 'False'; ExternalVisible := 'False'; ExternalWritable := 'False'; S7_SetPoint := 'True'} : TOF_TIME;   // Timer
      TimerHMICmdActivated { ExternalAccessible := 'False'; ExternalVisible := 'False'; ExternalWritable := 'False'; S7_SetPoint := 'True'} : TON_TIME;   // Timer
      TimerHMICmdDeactivated { ExternalAccessible := 'False'; ExternalVisible := 'False'; ExternalWritable := 'False'; S7_SetPoint := 'True'} : TON_TIME;   // Timer
   END_VAR
BEGIN

NETWORK
TITLE = **** 1 - Inputs **** DB number
// DB number
      L     DINO;
      T     #DBnr;

NETWORK
TITLE = **** 1 - Inputs **** Alarm class
// Alarm class
// Alarm class = E
      L     #I_AlarmClass;
      L     'E';
      ==I;
      =     #AlarmClass_E;

// Alarm class = D
      L     #I_AlarmClass;
      L     'D';
      ==I;
      =     #AlarmClass_D;

// Alarm class = C
      L     #I_AlarmClass;
      L     'C';
      ==I;
      =     #AlarmClass_C;

// Alarm class = B
      L     #I_AlarmClass;
      L     'B';
      ==I;
      =     #AlarmClass_B;

// Alarm class = A
      AN    #AlarmClass_B;
      AN    #AlarmClass_C;
      AN    #AlarmClass_D;
      AN    #AlarmClass_E;
      =     #AlarmClass_A;


REGION Network 3: **** 1 - Inputs **** HMI Cmd
   // Extract HMI Cmd
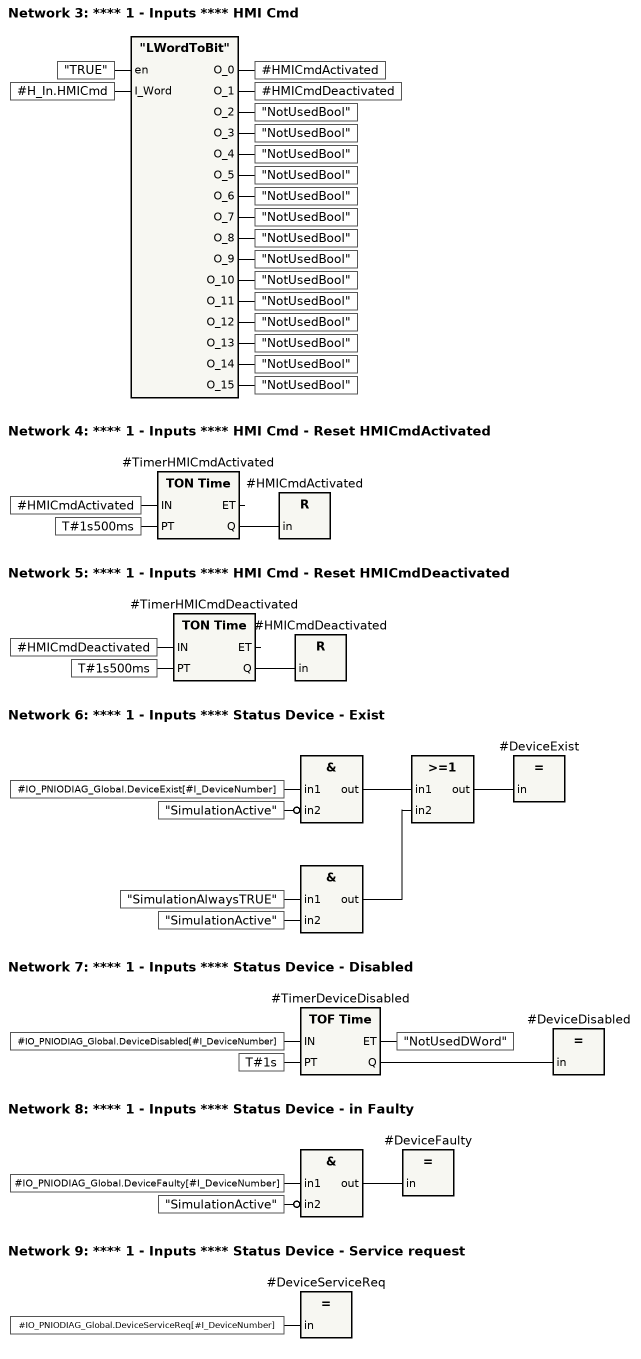
   IF "TRUE" THEN
       "LWordToBit"(I_Word := #H_In.HMICmd,
                    O_0 => #HMICmdActivated,
                    O_1 => #HMICmdDeactivated,
                    O_2 => "NotUsedBool",
                    O_3 => "NotUsedBool",
                    O_4 => "NotUsedBool",
                    O_5 => "NotUsedBool",
                    O_6 => "NotUsedBool",
                    O_7 => "NotUsedBool",
                    O_8 => "NotUsedBool",
                    O_9 => "NotUsedBool",
                    O_10 => "NotUsedBool",
                    O_11 => "NotUsedBool",
                    O_12 => "NotUsedBool",
                    O_13 => "NotUsedBool",
                    O_14 => "NotUsedBool",
                    O_15 => "NotUsedBool");
   END_IF;
END_REGION

REGION Network 4: **** 1 - Inputs **** HMI Cmd - Reset HMICmdActivated
   // HMI Cmd - Reset HMICmdActivated
   #TimerHMICmdActivated(IN := #HMICmdActivated, PT := T#1s500ms);   // TON
   IF #TimerHMICmdActivated.Q THEN #HMICmdActivated := FALSE; END_IF;
END_REGION

REGION Network 5: **** 1 - Inputs **** HMI Cmd - Reset HMICmdDeactivated
   // HMI Cmd - Reset HMICmdDeactivated
   #TimerHMICmdDeactivated(IN := #HMICmdDeactivated, PT := T#1s500ms);   // TON
   IF #TimerHMICmdDeactivated.Q THEN #HMICmdDeactivated := FALSE; END_IF;
END_REGION

REGION Network 6: **** 1 - Inputs **** Status Device - Exist
   // Status Device - Exist
   #DeviceExist := (#IO_PNIODIAG_Global.DeviceExist[#I_DeviceNumber] AND NOT "SimulationActive") OR ("SimulationAlwaysTRUE" AND "SimulationActive");
END_REGION

REGION Network 7: **** 1 - Inputs **** Status Device - Disabled
   // Status Device - Disabled
   #TimerDeviceDisabled(IN := #IO_PNIODIAG_Global.DeviceDisabled[#I_DeviceNumber],   // TOF
                        PT := T#1s,
                        ET => "NotUsedDWord");
   #DeviceDisabled := #TimerDeviceDisabled.Q;
END_REGION

REGION Network 8: **** 1 - Inputs **** Status Device - in Faulty
   // Status Device - in Faulty
   #DeviceFaulty := #IO_PNIODIAG_Global.DeviceFaulty[#I_DeviceNumber] AND NOT "SimulationActive";
END_REGION

REGION Network 9: **** 1 - Inputs **** Status Device - Service request
   // Status Device - Service request
   #DeviceServiceReq := #IO_PNIODIAG_Global.DeviceServiceReq[#I_DeviceNumber];
END_REGION

REGION Network 10: **** 1 - Inputs **** Timer Signal ActivateDeactivateBusy
   // Timer Signal ActivateDeactivateBusy
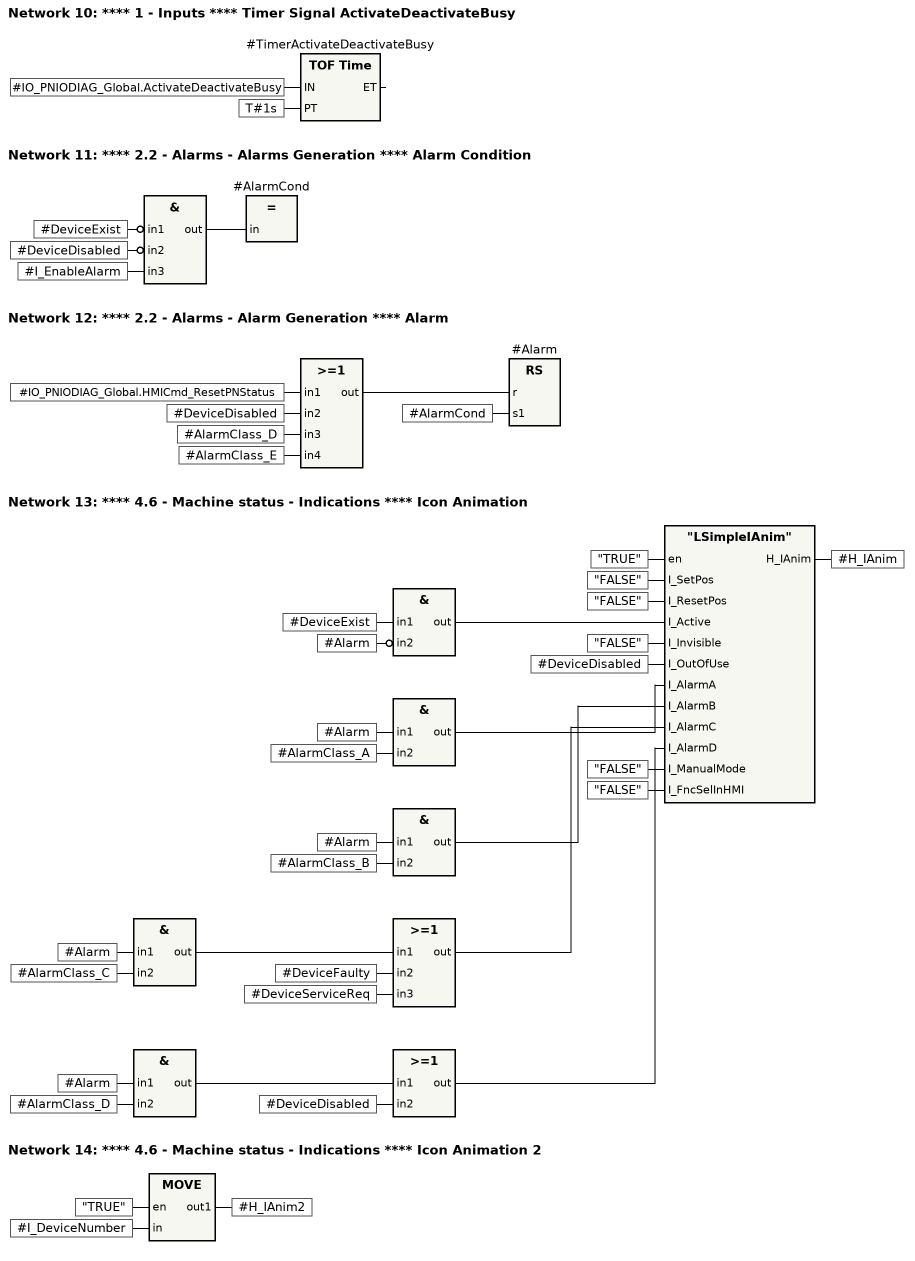
   #TimerActivateDeactivateBusy(IN := #IO_PNIODIAG_Global.ActivateDeactivateBusy, PT := T#1s);   // TOF
END_REGION

REGION Network 11: **** 2.2 - Alarms - Alarms Generation **** Alarm Condition
   // Condition for the Alarm
   #AlarmCond := NOT #DeviceExist AND NOT #DeviceDisabled AND #I_EnableAlarm;
END_REGION

REGION Network 12: **** 2.2 - Alarms - Alarm Generation **** Alarm
   // Alarm
   IF #IO_PNIODIAG_Global.HMICmd_ResetPNStatus OR #DeviceDisabled OR #AlarmClass_D OR #AlarmClass_E THEN
       #Alarm := FALSE;   // RS flip-flop
   END_IF;
   IF #AlarmCond THEN #Alarm := TRUE; END_IF;
END_REGION

REGION Network 13: **** 4.6 - Machine status - Indications **** Icon Animation
   // Icon Animation
   IF "TRUE" THEN
       "LSimpleIAnim"(I_SetPos := "FALSE",
                      I_ResetPos := "FALSE",
                      I_Active := #DeviceExist AND NOT #Alarm,
                      I_Invisible := "FALSE",
                      I_OutOfUse := #DeviceDisabled,
                      I_AlarmA := #Alarm AND #AlarmClass_A,
                      I_AlarmB := #Alarm AND #AlarmClass_B,
                      I_AlarmC := (#Alarm AND #AlarmClass_C) OR #DeviceFaulty OR #DeviceServiceReq,
                      I_AlarmD := (#Alarm AND #AlarmClass_D) OR #DeviceDisabled,
                      I_ManualMode := "FALSE",
                      I_FncSelInHMI := "FALSE",
                      H_IAnim => #H_IAnim);
   END_IF;
END_REGION

REGION Network 14: **** 4.6 - Machine status - Indications **** Icon Animation 2
   // Icon Animation Device number
   IF "TRUE" THEN #H_IAnim2 := #I_DeviceNumber; END_IF;
END_REGION

REGION Network 15: **** 4.6 - Machine status - Indications **** Animation
   // Animation for HMI
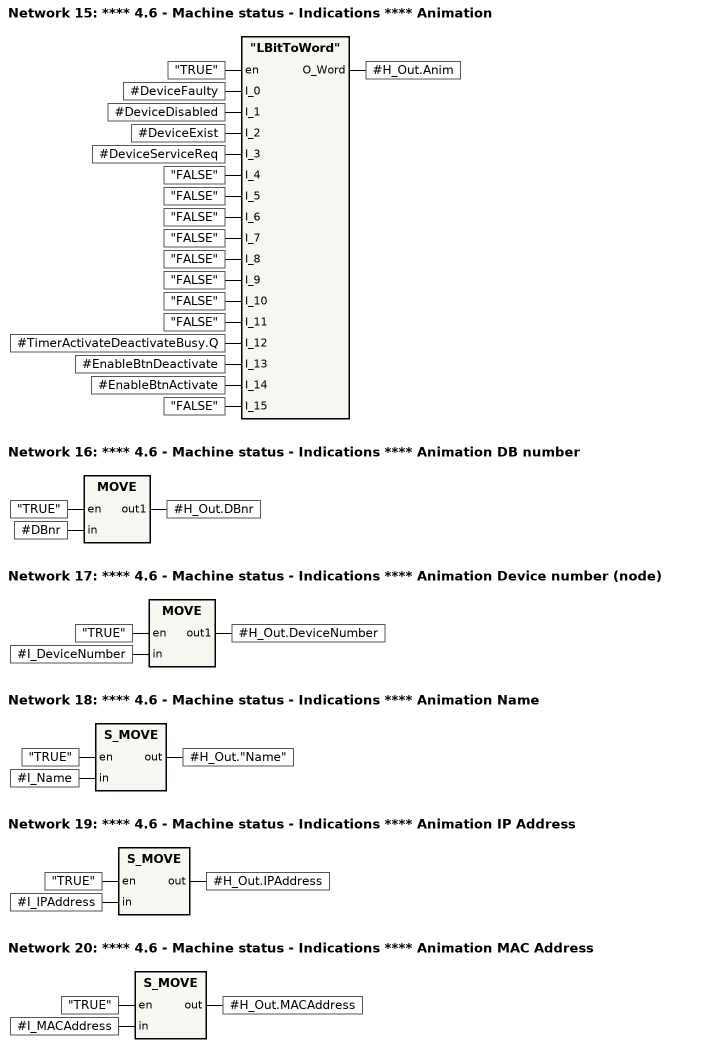
   IF "TRUE" THEN
       "LBitToWord"(I_0 := #DeviceFaulty,
                    I_1 := #DeviceDisabled,
                    I_2 := #DeviceExist,
                    I_3 := #DeviceServiceReq,
                    I_4 := "FALSE",
                    I_5 := "FALSE",
                    I_6 := "FALSE",
                    I_7 := "FALSE",
                    I_8 := "FALSE",
                    I_9 := "FALSE",
                    I_10 := "FALSE",
                    I_11 := "FALSE",
                    I_12 := #TimerActivateDeactivateBusy.Q,
                    I_13 := #EnableBtnDeactivate,
                    I_14 := #EnableBtnActivate,
                    I_15 := "FALSE",
                    O_Word => #H_Out.Anim);
   END_IF;
END_REGION

REGION Network 16: **** 4.6 - Machine status - Indications **** Animation DB number
   // DB number
   IF "TRUE" THEN #H_Out.DBnr := #DBnr; END_IF;
END_REGION

REGION Network 17: **** 4.6 - Machine status - Indications **** Animation Device number (node)
   // Device number (node)
   IF "TRUE" THEN #H_Out.DeviceNumber := #I_DeviceNumber; END_IF;
END_REGION

REGION Network 18: **** 4.6 - Machine status - Indications **** Animation Name
   // Name
   IF "TRUE" THEN #H_Out."Name" := #I_Name; END_IF;
END_REGION

REGION Network 19: **** 4.6 - Machine status - Indications **** Animation IP Address
   // IP Address
   IF "TRUE" THEN #H_Out.IPAddress := #I_IPAddress; END_IF;
END_REGION

REGION Network 20: **** 4.6 - Machine status - Indications **** Animation MAC Address
   // MAC Address
   IF "TRUE" THEN #H_Out.MACAddress := #I_MACAddress; END_IF;
END_REGION

REGION Network 21: **** 5.2 - Equations - Flow **** Activated or Deactived a device to the global FB
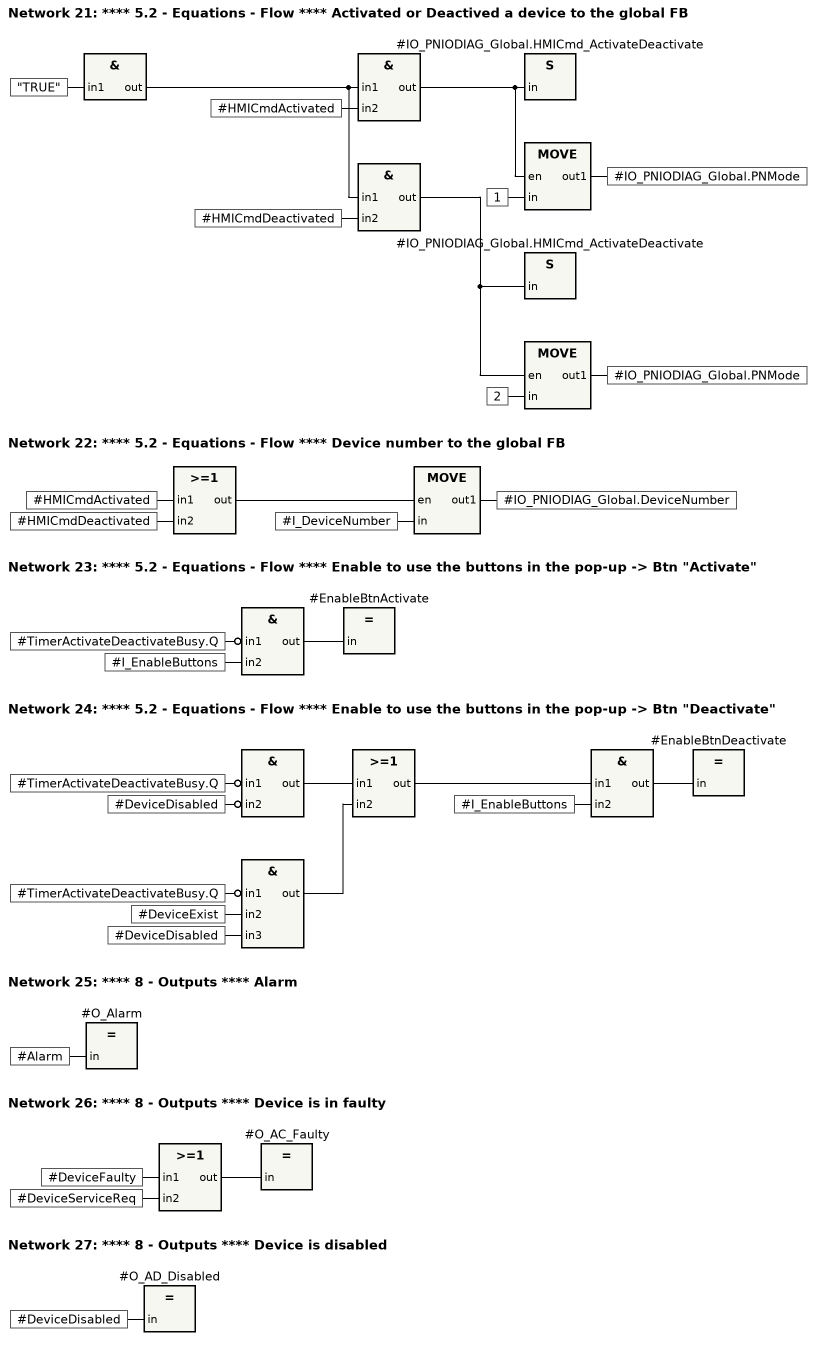
   IF "TRUE" AND #HMICmdActivated THEN
       #IO_PNIODIAG_Global.HMICmd_ActivateDeactivate := TRUE;
       #IO_PNIODIAG_Global.PNMode := 1;
   END_IF;
   IF "TRUE" AND #HMICmdDeactivated THEN
       #IO_PNIODIAG_Global.HMICmd_ActivateDeactivate := TRUE;
       #IO_PNIODIAG_Global.PNMode := 2;
   END_IF;
END_REGION

REGION Network 22: **** 5.2 - Equations - Flow **** Device number to the global FB
   IF #HMICmdActivated OR #HMICmdDeactivated THEN
       #IO_PNIODIAG_Global.DeviceNumber := #I_DeviceNumber;
   END_IF;
END_REGION

REGION Network 23: **** 5.2 - Equations - Flow **** Enable to use the buttons in the pop-up -> Btn "Activate"
   // Enable to use the buttons in the pop-up -> Btn "Activate"
   #EnableBtnActivate := NOT #TimerActivateDeactivateBusy.Q AND #I_EnableButtons;
END_REGION

REGION Network 24: **** 5.2 - Equations - Flow **** Enable to use the buttons in the pop-up -> Btn "Deactivate"
   // Enable to use the buttons in the pop-up -> Btn "Deactivate"
   #EnableBtnDeactivate := ((NOT #TimerActivateDeactivateBusy.Q AND NOT #DeviceDisabled) OR (NOT #TimerActivateDeactivateBusy.Q AND #DeviceExist AND #DeviceDisabled)) AND #I_EnableButtons;
END_REGION

REGION Network 25: **** 8 - Outputs **** Alarm
   // Alarm
   #O_Alarm := #Alarm;
END_REGION

REGION Network 26: **** 8 - Outputs **** Device is in faulty
   #O_AC_Faulty := #DeviceFaulty OR #DeviceServiceReq;
END_REGION

REGION Network 27: **** 8 - Outputs **** Device is disabled
   #O_AD_Disabled := #DeviceDisabled;
END_REGION

REGION Network 28: **** 8 - Outputs **** Alarm AB Condition
   // Alarm AB condition
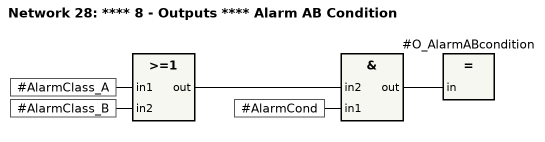
   #O_AlarmABcondition := (#AlarmClass_A OR #AlarmClass_B) AND #AlarmCond;
END_REGION
END_FUNCTION_BLOCK

FUNCTION_BLOCK "LPhoneAlarmReqString"   // FB2255, FBD
TITLE = LPhoneAlarmReq
{ S7_Optimized_Access := 'FALSE' }
AUTHOR : VCC
FAMILY : Function
VERSION : 0.1
// =============================================================================
// This Module Handles Phone Alarm Requests
// =============================================================================
// stored: AutoNumber false, IsIECCheckEnabled false, SetENOAutomatically False, UDAEnableTagReadback false
   VAR_INPUT
      I_PhoneAlarmReq1 { ExternalAccessible := 'False'; ExternalVisible := 'False'; ExternalWritable := 'False'} : Bool;   // Request Team Leader Andon From Loading Stn / Request PhoneAlarm For Station / Request PhoneAlarm
      I_PhoneAlarmReq2 { ExternalAccessible := 'False'; ExternalVisible := 'False'; ExternalWritable := 'False'} : Bool;   // Request Maintenance Andon From Loading Stn / Request PhoneAlarm For Station / Request PhoneAlarm
      I_PhoneAlarmReq3 { ExternalAccessible := 'False'; ExternalVisible := 'False'; ExternalWritable := 'False'} : Bool;   // Request PhoneAlarm For Station / Request PhoneAlarm
      I_PhoneAlarmReq4 { ExternalAccessible := 'False'; ExternalVisible := 'False'; ExternalWritable := 'False'} : Bool;   // Request PhoneAlarm For Station / Request PhoneAlarm
      I_PhoneAlarmReq5 { ExternalAccessible := 'False'; ExternalVisible := 'False'; ExternalWritable := 'False'} : Bool;   // Request PhoneAlarm For Station / Request PhoneAlarm
      I_PhoneAlarmReq6 { ExternalAccessible := 'False'; ExternalVisible := 'False'; ExternalWritable := 'False'} : Bool;   // Request PhoneAlarm For Station / Request PhoneAlarm
      I_PhoneAlarmReq7 { ExternalAccessible := 'False'; ExternalVisible := 'False'; ExternalWritable := 'False'} : Bool;   // Request PhoneAlarm For Station / Request PhoneAlarm
      I_PhoneAlarmReq8 { ExternalAccessible := 'False'; ExternalVisible := 'False'; ExternalWritable := 'False'} : Bool;   // Request PhoneAlarm For Station / Request PhoneAlarm
      I_PhoneAlarmReq9 { ExternalAccessible := 'False'; ExternalVisible := 'False'; ExternalWritable := 'False'} : Bool;   // Request PhoneAlarm For Station / Request PhoneAlarm
      I_PhoneAlarmReq10 { ExternalAccessible := 'False'; ExternalVisible := 'False'; ExternalWritable := 'False'} : Bool;   // Request PhoneAlarm For Station / Request PhoneAlarm
      I_PhoneAlarmReq11 { ExternalAccessible := 'False'; ExternalVisible := 'False'; ExternalWritable := 'False'} : Bool;   // Request PhoneAlarm For Station / Request PhoneAlarm
      I_PhoneAlarmReq12 { ExternalAccessible := 'False'; ExternalVisible := 'False'; ExternalWritable := 'False'} : Bool;   // Request PhoneAlarm For Station / Request PhoneAlarm
      I_PhoneAlarmReq13 { ExternalAccessible := 'False'; ExternalVisible := 'False'; ExternalWritable := 'False'} : Bool;   // Request PhoneAlarm For Station / Request PhoneAlarm
      I_PhoneAlarmReq14 { ExternalAccessible := 'False'; ExternalVisible := 'False'; ExternalWritable := 'False'} : Bool;   // Request PhoneAlarm For Station / Request PhoneAlarm
      I_PhoneAlarmReq15 { ExternalAccessible := 'False'; ExternalVisible := 'False'; ExternalWritable := 'False'} : Bool;   // Request PhoneAlarm For Station / Request PhoneAlarm
      I_PhoneAlarmReq16 { ExternalAccessible := 'False'; ExternalVisible := 'False'; ExternalWritable := 'False'} : Bool;   // Request PhoneAlarm For Station / Request PhoneAlarm
      C_MessageType1 { ExternalAccessible := 'False'; ExternalVisible := 'False'; ExternalWritable := 'False'} : String[20];   // Configuration Station / Configuration Message
      C_Message1 { ExternalAccessible := 'False'; ExternalVisible := 'False'; ExternalWritable := 'False'} : String[120];   // Configuration Station / Configuration Message
      C_MessageType2 { ExternalAccessible := 'False'; ExternalVisible := 'False'; ExternalWritable := 'False'} : String[20];   // Configuration Station / Configuration Message
      C_Message2 { ExternalAccessible := 'False'; ExternalVisible := 'False'; ExternalWritable := 'False'} : String[120];   // Configuration Station / Configuration Message
      C_MessageType3 { ExternalAccessible := 'False'; ExternalVisible := 'False'; ExternalWritable := 'False'} : String[20];   // Configuration Station / Configuration Message
      C_Message3 { ExternalAccessible := 'False'; ExternalVisible := 'False'; ExternalWritable := 'False'} : String[120];   // Configuration Station / Configuration Message
      C_MessageType4 { ExternalAccessible := 'False'; ExternalVisible := 'False'; ExternalWritable := 'False'} : String[20];   // Configuration Station / Configuration Message
      C_Message4 { ExternalAccessible := 'False'; ExternalVisible := 'False'; ExternalWritable := 'False'} : String[120];   // Configuration Station / Configuration Message
      C_MessageType5 { ExternalAccessible := 'False'; ExternalVisible := 'False'; ExternalWritable := 'False'} : String[20];   // Configuration Station / Configuration Message
      C_Message5 { ExternalAccessible := 'False'; ExternalVisible := 'False'; ExternalWritable := 'False'} : String[120];   // Configuration Station / Configuration Message
      C_MessageType6 { ExternalAccessible := 'False'; ExternalVisible := 'False'; ExternalWritable := 'False'} : String[20];   // Configuration Station / Configuration Message
      C_Message6 { ExternalAccessible := 'False'; ExternalVisible := 'False'; ExternalWritable := 'False'} : String[120];   // Configuration Station / Configuration Message
      C_MessageType7 { ExternalAccessible := 'False'; ExternalVisible := 'False'; ExternalWritable := 'False'} : String[20];   // Configuration Station / Configuration Message
      C_Message7 { ExternalAccessible := 'False'; ExternalVisible := 'False'; ExternalWritable := 'False'} : String[120];   // Configuration Station / Configuration Message
      C_MessageType8 { ExternalAccessible := 'False'; ExternalVisible := 'False'; ExternalWritable := 'False'} : String[20];   // Configuration Station / Configuration Message
      C_Message8 { ExternalAccessible := 'False'; ExternalVisible := 'False'; ExternalWritable := 'False'} : String[120];   // Configuration Station / Configuration Message
      C_MessageType9 { ExternalAccessible := 'False'; ExternalVisible := 'False'; ExternalWritable := 'False'} : String[20];   // Configuration Station / Configuration Message
      C_Message9 { ExternalAccessible := 'False'; ExternalVisible := 'False'; ExternalWritable := 'False'} : String[120];   // Configuration Station / Configuration Message
      C_MessageType10 { ExternalAccessible := 'False'; ExternalVisible := 'False'; ExternalWritable := 'False'} : String[20];   // Configuration Station / Configuration Message
      C_Message10 { ExternalAccessible := 'False'; ExternalVisible := 'False'; ExternalWritable := 'False'} : String[120];   // Configuration Station / Configuration Message
      C_MessageType11 { ExternalAccessible := 'False'; ExternalVisible := 'False'; ExternalWritable := 'False'} : String[20];   // Configuration Station / Configuration Message
      C_Message11 { ExternalAccessible := 'False'; ExternalVisible := 'False'; ExternalWritable := 'False'} : String[120];   // Configuration Station / Configuration Message
      C_MessageType12 { ExternalAccessible := 'False'; ExternalVisible := 'False'; ExternalWritable := 'False'} : String[20];   // Configuration Station / Configuration Message
      C_Message12 { ExternalAccessible := 'False'; ExternalVisible := 'False'; ExternalWritable := 'False'} : String[120];   // Configuration Station / Configuration Message
      C_MessageType13 { ExternalAccessible := 'False'; ExternalVisible := 'False'; ExternalWritable := 'False'} : String[20];   // Configuration Station / Configuration Message
      C_Message13 { ExternalAccessible := 'False'; ExternalVisible := 'False'; ExternalWritable := 'False'} : String[120];   // Configuration Station / Configuration Message
      C_MessageType14 { ExternalAccessible := 'False'; ExternalVisible := 'False'; ExternalWritable := 'False'} : String[20];   // Configuration Station / Configuration Message
      C_Message14 { ExternalAccessible := 'False'; ExternalVisible := 'False'; ExternalWritable := 'False'} : String[120];   // Configuration Station / Configuration Message
      C_MessageType15 { ExternalAccessible := 'False'; ExternalVisible := 'False'; ExternalWritable := 'False'} : String[20];   // Configuration Station / Configuration Message
      C_Message15 { ExternalAccessible := 'False'; ExternalVisible := 'False'; ExternalWritable := 'False'} : String[120];   // Configuration Station / Configuration Message
      C_MessageType16 { ExternalAccessible := 'False'; ExternalVisible := 'False'; ExternalWritable := 'False'} : String[20];   // Configuration Station / Configuration Message
      C_Message16 { ExternalAccessible := 'False'; ExternalVisible := 'False'; ExternalWritable := 'False'} : String[120];   // Configuration Station / Configuration Message
      C_VDCommRecvDB { ExternalAccessible := 'False'; ExternalVisible := 'False'; ExternalWritable := 'False'} : DB_ANY;   // VD communication system receive DB; Not to be used by application / VD communication system receive DB Not to be used by Application
      C_VDCommSendDB { ExternalAccessible := 'False'; ExternalVisible := 'False'; ExternalWritable := 'False'} : DB_ANY;   // VD communication system send DB; Not to be used by application / VD communication system send DB Not to be used by Application
      C_LocalRecvDB { ExternalAccessible := 'False'; ExternalVisible := 'False'; ExternalWritable := 'False'} : DB_ANY;   // Local DB To Store Received Data
      C_LocalSendDB { ExternalAccessible := 'False'; ExternalVisible := 'False'; ExternalWritable := 'False'} : DB_ANY;   // Local DB for send data; to be used by application / Local DB For Send Data Used By The Application
      C_SubSystem { ExternalAccessible := 'False'; ExternalVisible := 'False'; ExternalWritable := 'False'} : Int;   // Number to identify the subsystem / Identify Subsystem
      C_FilterMessage1 { ExternalAccessible := 'False'; ExternalVisible := 'False'; ExternalWritable := 'False'} : Time;   // Filter
      C_FilterMessage2 { ExternalAccessible := 'False'; ExternalVisible := 'False'; ExternalWritable := 'False'} : Time;   // Filter
      C_FilterMessage3 { ExternalAccessible := 'False'; ExternalVisible := 'False'; ExternalWritable := 'False'} : Time;   // Filter
      C_FilterMessage4 { ExternalAccessible := 'False'; ExternalVisible := 'False'; ExternalWritable := 'False'} : Time;   // Filter
      C_FilterMessage5 { ExternalAccessible := 'False'; ExternalVisible := 'False'; ExternalWritable := 'False'} : Time;   // Filter
      C_FilterMessage6 { ExternalAccessible := 'False'; ExternalVisible := 'False'; ExternalWritable := 'False'} : Time;   // Filter
      C_FilterMessage7 { ExternalAccessible := 'False'; ExternalVisible := 'False'; ExternalWritable := 'False'} : Time;   // Filter
      C_FilterMessage8 { ExternalAccessible := 'False'; ExternalVisible := 'False'; ExternalWritable := 'False'} : Time;   // Filter
      C_FilterMessage9 { ExternalAccessible := 'False'; ExternalVisible := 'False'; ExternalWritable := 'False'} : Time;   // Filter
      C_FilterMessage10 { ExternalAccessible := 'False'; ExternalVisible := 'False'; ExternalWritable := 'False'} : Time;   // Filter
      C_FilterMessage11 { ExternalAccessible := 'False'; ExternalVisible := 'False'; ExternalWritable := 'False'} : Time;   // Filter
      C_FilterMessage12 { ExternalAccessible := 'False'; ExternalVisible := 'False'; ExternalWritable := 'False'} : Time;   // Filter
      C_FilterMessage13 { ExternalAccessible := 'False'; ExternalVisible := 'False'; ExternalWritable := 'False'} : Time;   // Filter
      C_FilterMessage14 { ExternalAccessible := 'False'; ExternalVisible := 'False'; ExternalWritable := 'False'} : Time;   // Filter
      C_FilterMessage15 { ExternalAccessible := 'False'; ExternalVisible := 'False'; ExternalWritable := 'False'} : Time;   // Filter
      C_FilterMessage16 { ExternalAccessible := 'False'; ExternalVisible := 'False'; ExternalWritable := 'False'} : Time;   // Filter
   END_VAR
   VAR_IN_OUT
      IO_VD : "VDComm";   // Communication
      H_HMI : "H_HMI";   // Animation
      H_PhoneAlarmReqString : "H_PhoneAlarmReqString";   // Animation
   END_VAR
   VAR DB_SPECIFIC
      ReqPhoneAlarm { ExternalAccessible := 'False'; ExternalVisible := 'False'; ExternalWritable := 'False'} : Array[1..16] of Bool;   // Request Team Leader Andon / Request PhoneAlarm
      VDReqPhoneAlarm { ExternalAccessible := 'False'; ExternalVisible := 'False'; ExternalWritable := 'False'} : Array[1..16] of Bool;   // VD Request Team Leader Andon / VD Request PhoneAlarm
      Done { ExternalAccessible := 'False'; ExternalVisible := 'False'; ExternalWritable := 'False'} : Array[1..16] of Bool;   // Array
      StnEdge { ExternalAccessible := 'False'; ExternalVisible := 'False'; ExternalWritable := 'False'} : Array[1..16] of Bool;   // Pos Edge
      SendDoneToVD { ExternalAccessible := 'False'; ExternalVisible := 'False'; ExternalWritable := 'False'} : Bool;   // Request Is Finished
      SendVD { ExternalAccessible := 'False'; ExternalVisible := 'False'; ExternalWritable := 'False'} : Bool;   // Send
      PhoneAlarmReqActiveStn1 { ExternalAccessible := 'False'; ExternalVisible := 'False'; ExternalWritable := 'False'} : Bool;   // Indication Request Team Leader Andon / Indication Request
      PhoneAlarmReqActiveStn2 { ExternalAccessible := 'False'; ExternalVisible := 'False'; ExternalWritable := 'False'} : Bool;   // Indication Maintenance Andon / Indication Request
      PhoneAlarmReqActiveStn3 { ExternalAccessible := 'False'; ExternalVisible := 'False'; ExternalWritable := 'False'} : Bool;   // Indication Request
      PhoneAlarmReqActiveStn4 { ExternalAccessible := 'False'; ExternalVisible := 'False'; ExternalWritable := 'False'} : Bool;   // Indication Request
      PhoneAlarmReqActiveStn5 { ExternalAccessible := 'False'; ExternalVisible := 'False'; ExternalWritable := 'False'} : Bool;   // Indication Request
      PhoneAlarmReqActiveStn6 { ExternalAccessible := 'False'; ExternalVisible := 'False'; ExternalWritable := 'False'} : Bool;   // Indication Request
      PhoneAlarmReqActiveStn7 { ExternalAccessible := 'False'; ExternalVisible := 'False'; ExternalWritable := 'False'} : Bool;   // Indication Request
      PhoneAlarmReqActiveStn8 { ExternalAccessible := 'False'; ExternalVisible := 'False'; ExternalWritable := 'False'} : Bool;   // Indication Request
      PhoneAlarmReqActiveStn9 { ExternalAccessible := 'False'; ExternalVisible := 'False'; ExternalWritable := 'False'} : Bool;   // Indication Request
      PhoneAlarmReqActiveStn10 { ExternalAccessible := 'False'; ExternalVisible := 'False'; ExternalWritable := 'False'} : Bool;   // Indication Request
      PhoneAlarmReqActiveStn11 { ExternalAccessible := 'False'; ExternalVisible := 'False'; ExternalWritable := 'False'} : Bool;   // Indication Request
      PhoneAlarmReqActiveStn12 { ExternalAccessible := 'False'; ExternalVisible := 'False'; ExternalWritable := 'False'} : Bool;   // Indication Request
      PhoneAlarmReqActiveStn13 { ExternalAccessible := 'False'; ExternalVisible := 'False'; ExternalWritable := 'False'} : Bool;   // Indication Request
      PhoneAlarmReqActiveStn14 { ExternalAccessible := 'False'; ExternalVisible := 'False'; ExternalWritable := 'False'} : Bool;   // Indication Request
      PhoneAlarmReqActiveStn15 { ExternalAccessible := 'False'; ExternalVisible := 'False'; ExternalWritable := 'False'} : Bool;   // Indication Request
      PhoneAlarmReqActiveStn16 { ExternalAccessible := 'False'; ExternalVisible := 'False'; ExternalWritable := 'False'} : Bool;   // Indication Request
      VDMessage { ExternalAccessible := 'False'; ExternalVisible := 'False'; ExternalWritable := 'False'} : Struct   // VD MEssage to send
         VDMessageType { ExternalAccessible := 'False'; ExternalVisible := 'False'; ExternalWritable := 'False'} : Array[0..19] of Byte;   // Attention Event / VD MessageType
         VDMessage { ExternalAccessible := 'False'; ExternalVisible := 'False'; ExternalWritable := 'False'} : Array[0..119] of Byte;   // Attention Event / VD Message
      END_STRUCT;
   END_VAR
   VAR
      _VDComSubSystem { ExternalAccessible := 'False'; ExternalVisible := 'False'; ExternalWritable := 'False'; S7_SetPoint := 'True'} : "LVDComSubSystemS7-1500";   // FB
   END_VAR
   VAR DB_SPECIFIC
      Edge { ExternalAccessible := 'False'; ExternalVisible := 'False'; ExternalWritable := 'False'} : Array[0..15] of Bool;   // Array Edge
      InitDone { ExternalAccessible := 'False'; ExternalVisible := 'False'; ExternalWritable := 'False'} : Array[1..32] of Bool;   // Init Done
      InitDoneEdge { ExternalAccessible := 'False'; ExternalVisible := 'False'; ExternalWritable := 'False'} : Array[1..32] of Bool;   // Edge Done
      MessageType { ExternalAccessible := 'False'; ExternalVisible := 'False'; ExternalWritable := 'False'} : Int;   // Message Type
      MessageLength { ExternalAccessible := 'False'; ExternalVisible := 'False'; ExternalWritable := 'False'} : Word;   // Message Type / Message Lenght
      _Filter1 { ExternalAccessible := 'False'; ExternalVisible := 'False'; ExternalWritable := 'False'; S7_SetPoint := 'True'} : TON_TIME;   // FB
      _Filter2 { ExternalAccessible := 'False'; ExternalVisible := 'False'; ExternalWritable := 'False'; S7_SetPoint := 'True'} : TON_TIME;   // FB
      _Filter3 { ExternalAccessible := 'False'; ExternalVisible := 'False'; ExternalWritable := 'False'; S7_SetPoint := 'True'} : TON_TIME;   // FB
      _Filter4 { ExternalAccessible := 'False'; ExternalVisible := 'False'; ExternalWritable := 'False'; S7_SetPoint := 'True'} : TON_TIME;   // FB
      _Filter5 { ExternalAccessible := 'False'; ExternalVisible := 'False'; ExternalWritable := 'False'; S7_SetPoint := 'True'} : TON_TIME;   // FB
      _Filter6 { ExternalAccessible := 'False'; ExternalVisible := 'False'; ExternalWritable := 'False'; S7_SetPoint := 'True'} : TON_TIME;   // FB
      _Filter7 { ExternalAccessible := 'False'; ExternalVisible := 'False'; ExternalWritable := 'False'; S7_SetPoint := 'True'} : TON_TIME;   // FB
      _Filter8 { ExternalAccessible := 'False'; ExternalVisible := 'False'; ExternalWritable := 'False'; S7_SetPoint := 'True'} : TON_TIME;   // FB
      _Filter9 { ExternalAccessible := 'False'; ExternalVisible := 'False'; ExternalWritable := 'False'; S7_SetPoint := 'True'} : TON_TIME;   // FB
      _Filter10 { ExternalAccessible := 'False'; ExternalVisible := 'False'; ExternalWritable := 'False'; S7_SetPoint := 'True'} : TON_TIME;   // FB
      _Filter11 { ExternalAccessible := 'False'; ExternalVisible := 'False'; ExternalWritable := 'False'; S7_SetPoint := 'True'} : TON_TIME;   // FB
      _Filter12 { ExternalAccessible := 'False'; ExternalVisible := 'False'; ExternalWritable := 'False'; S7_SetPoint := 'True'} : TON_TIME;   // FB
      _Filter13 { ExternalAccessible := 'False'; ExternalVisible := 'False'; ExternalWritable := 'False'; S7_SetPoint := 'True'} : TON_TIME;   // FB
      _Filter14 { ExternalAccessible := 'False'; ExternalVisible := 'False'; ExternalWritable := 'False'; S7_SetPoint := 'True'} : TON_TIME;   // FB
      _Filter15 { ExternalAccessible := 'False'; ExternalVisible := 'False'; ExternalWritable := 'False'; S7_SetPoint := 'True'} : TON_TIME;   // FB
      _Filter16 { ExternalAccessible := 'False'; ExternalVisible := 'False'; ExternalWritable := 'False'; S7_SetPoint := 'True'} : TON_TIME;   // FB
      SendToVDTimeOut { ExternalAccessible := 'False'; ExternalVisible := 'False'; ExternalWritable := 'False'; S7_SetPoint := 'True'} : TON_TIME;   // Send to VD time-out
      ResetVDComm { ExternalAccessible := 'False'; ExternalVisible := 'False'; ExternalWritable := 'False'} : Bool;   // Reset VD communication upon timeout
      VDMessageTypeTemp { ExternalAccessible := 'False'; ExternalVisible := 'False'; ExternalWritable := 'False'} : String[20];   // Attention Event / VDMessageTypeTemp string 20 characters
      VDMessageTemp { ExternalAccessible := 'False'; ExternalVisible := 'False'; ExternalWritable := 'False'} : String[120];   // Attention Event / VDMessageTemp string 120 characters
      VDMessageTypeSerialzePos { ExternalAccessible := 'False'; ExternalVisible := 'False'; ExternalWritable := 'False'} : DInt;   // Serialize position
      VDMessageSerialzePos { ExternalAccessible := 'False'; ExternalVisible := 'False'; ExternalWritable := 'False'} : DInt;   // Serialize position
      VDMessageTypeTempArray { ExternalAccessible := 'False'; ExternalVisible := 'False'; ExternalWritable := 'False'} : Array[0..21] of Byte;   // VDMessageType Array
      VDMessageTempArray { ExternalAccessible := 'False'; ExternalVisible := 'False'; ExternalWritable := 'False'} : Array[0..121] of Byte;   // VDMessage Array
   END_VAR
   VAR_TEMP
      RequestCommand1 : Bool;   // Light On To Building Infrastructure / Request Configured Command
      RequestCommand2 : Bool;   // Light On To Building Infrastructure / Request Configured Command
      RequestCommand3 : Bool;   // Light On To Building Infrastructure / Request Configured Command
      RequestCommand4 : Bool;   // Light On To Building Infrastructure / Request Configured Command
      RequestCommand5 : Bool;   // Light On To Building Infrastructure / Request Configured Command
      RequestCommand6 : Bool;   // Light On To Building Infrastructure / Request Configured Command
      RequestCommand7 : Bool;   // Light On To Building Infrastructure / Request Configured Command
      RequestCommand8 : Bool;   // Light On To Building Infrastructure / Request Configured Command
      RequestCommand9 : Bool;   // Request Configured Command
      RequestCommand10 : Bool;   // Request Configured Command
      RequestCommand11 : Bool;   // Request Configured Command
      RequestCommand12 : Bool;   // Request Configured Command
      RequestCommand13 : Bool;   // Request Configured Command
      RequestCommand14 : Bool;   // Request Configured Command
      RequestCommand15 : Bool;   // Request Configured Command
      RequestCommand16 : Bool;   // Request Configured Command
      RecvDBNbr : Int;   // Receive system DB Number
      SendDBNbr : Int;   // Send system DB Number
      LocalRecvDBNbr : Int;   // Receive DB Number Local by Application
      LocalSendDBNbr : Int;   // Send DB Number Local by Application
      PtrASnd : Any;   // Pointer to the Application receive DB / Pointer to the Application send DB
   END_VAR
   VAR CONSTANT
      String20Spaces : String := '                    ';   // String with 20 spaces
      String120Spaces : String := '                                                                                                                        ';   // String with 120 spaces
   END_VAR
   VAR_TEMP   // added for the SCL form of the ladder/FBD networks
      _w1 : Bool;
      _w2 : Bool;
   END_VAR
BEGIN

REGION Network 1: **** 1 - Inputs **** Extract The Commands From HMI
   // Extract The Commands From HMI
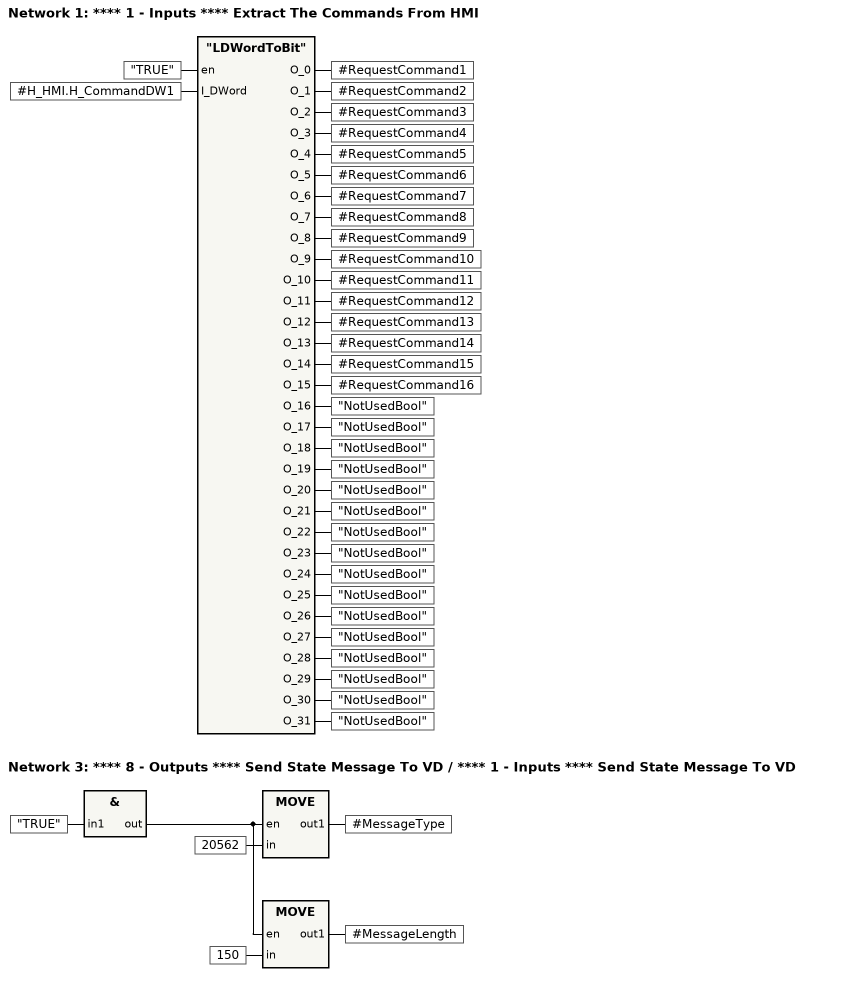
   IF "TRUE" THEN
       "LDWordToBit"(I_DWord := #H_HMI.H_CommandDW1,
                     O_0 => #RequestCommand1,
                     O_1 => #RequestCommand2,
                     O_2 => #RequestCommand3,
                     O_3 => #RequestCommand4,
                     O_4 => #RequestCommand5,
                     O_5 => #RequestCommand6,
                     O_6 => #RequestCommand7,
                     O_7 => #RequestCommand8,
                     O_8 => #RequestCommand9,
                     O_9 => #RequestCommand10,
                     O_10 => #RequestCommand11,
                     O_11 => #RequestCommand12,
                     O_12 => #RequestCommand13,
                     O_13 => #RequestCommand14,
                     O_14 => #RequestCommand15,
                     O_15 => #RequestCommand16,
                     O_16 => "NotUsedBool",
                     O_17 => "NotUsedBool",
                     O_18 => "NotUsedBool",
                     O_19 => "NotUsedBool",
                     O_20 => "NotUsedBool",
                     O_21 => "NotUsedBool",
                     O_22 => "NotUsedBool",
                     O_23 => "NotUsedBool",
                     O_24 => "NotUsedBool",
                     O_25 => "NotUsedBool",
                     O_26 => "NotUsedBool",
                     O_27 => "NotUsedBool",
                     O_28 => "NotUsedBool",
                     O_29 => "NotUsedBool",
                     O_30 => "NotUsedBool",
                     O_31 => "NotUsedBool");
   END_IF;
END_REGION

NETWORK
TITLE = **** 1 - Inputs **** Load DB / **** 1 - Inputs **** Load DB number
// Load DB numbers to local variables from the Receive and Send DB from - VD Master - VD Subsystem
// Read DB Number Recv
      OPN   #C_VDCommRecvDB;
      L     DBNO;
      T     #RecvDBNbr;

// Read DB Number Send
      OPN   #C_VDCommSendDB;
      L     DBNO;
      T     #SendDBNbr;

// DB Number from VD Sub system
      OPN   #C_LocalRecvDB;
      L     DBNO;
      T     #LocalRecvDBNbr;

// Read DB Number Send
      OPN   #C_LocalSendDB;
      L     DBNO;
      T     #LocalSendDBNbr;

REGION Network 3: **** 8 - Outputs **** Send State Message To VD / **** 1 - Inputs **** Send State Message To VD
   // Send State Message To VD
   IF "TRUE" THEN
       #MessageType := 20562;
       #MessageLength := 150;
   END_IF;
END_REGION

REGION Network 4: **** 3.1 - Communication - Other Systems **** Send Message
   // Send Message
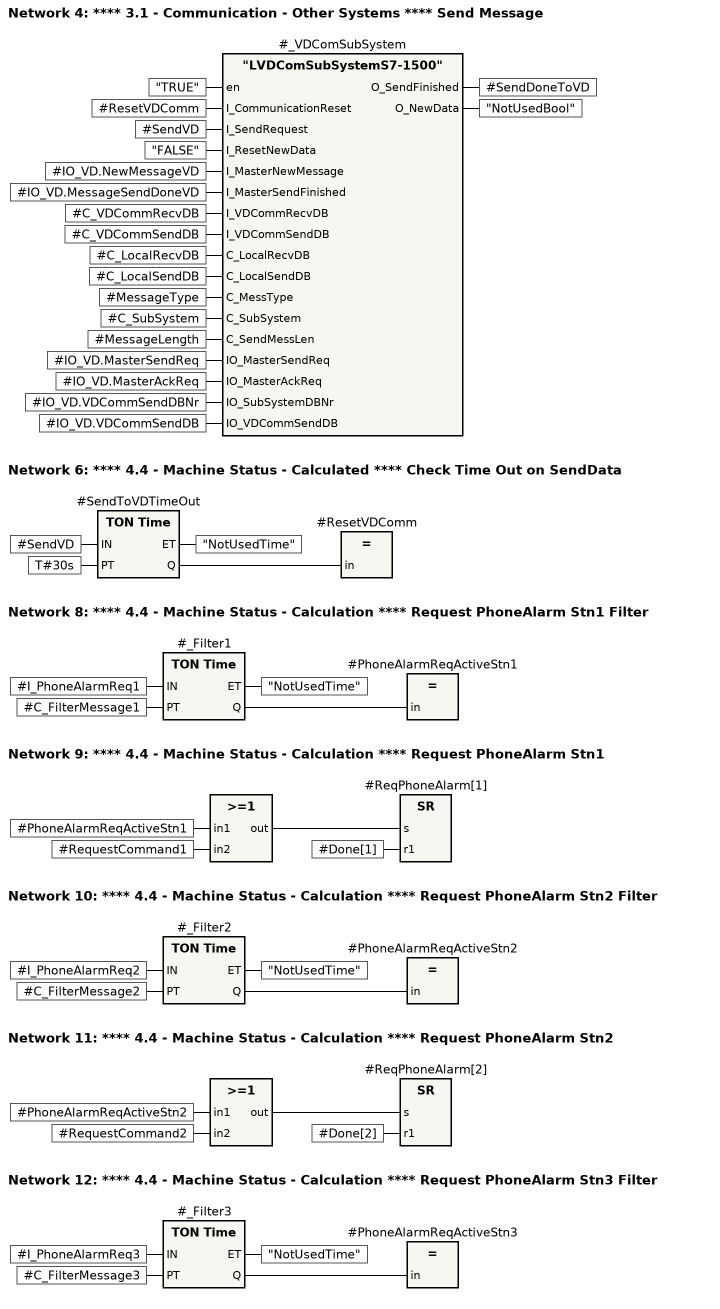
   IF "TRUE" THEN
       #_VDComSubSystem(I_CommunicationReset := #ResetVDComm,   // "LVDComSubSystemS7-1500"
                        I_SendRequest := #SendVD,
                        I_ResetNewData := "FALSE",
                        I_MasterNewMessage := #IO_VD.NewMessageVD,
                        I_MasterSendFinished := #IO_VD.MessageSendDoneVD,
                        I_VDCommRecvDB := #C_VDCommRecvDB,
                        I_VDCommSendDB := #C_VDCommSendDB,
                        C_LocalRecvDB := #C_LocalRecvDB,
                        C_LocalSendDB := #C_LocalSendDB,
                        C_MessType := #MessageType,
                        C_SubSystem := #C_SubSystem,
                        C_SendMessLen := #MessageLength,
                        IO_MasterSendReq := #IO_VD.MasterSendReq,
                        IO_MasterAckReq := #IO_VD.MasterAckReq,
                        IO_SubSystemDBNr := #IO_VD.VDCommSendDBNr,
                        IO_VDCommSendDB := #IO_VD.VDCommSendDB,
                        O_SendFinished => #SendDoneToVD,
                        O_NewData => "NotUsedBool");
   END_IF;
END_REGION

NETWORK
TITLE = **** 3.1 - Communication - Other Systems **** Configure DB / **** 4.2 Parameter **** Configure DB
// Configure DB pointers
      LAR1  P##PtrASnd;
      L     16#1002;  // Data type to copy B#16#2 = Bytes
      T     LW [AR1, P#0.0];
      L     #MessageLength;  //Length sending data
      T     LW [AR1, P#2.0];
      L     #LocalSendDBNbr;  // Local Send DB Number
      T     LW [AR1, P#4.0];
      L     10;  // Offset in DB (skip VD header)
      SLD   3;  // Convert to pointer - Shift Left DW
      OD    16#8400_0000;  // Memory area DB Memory - 84 equals DB
      T     LD [AR1, P#6.0];


REGION Network 6: **** 4.4 - Machine Status - Calculated **** Check Time Out on SendData
   // Reset Send request when time out elapses
   // Reset the VD communication
   #SendToVDTimeOut(IN := #SendVD, PT := T#30s, ET => "NotUsedTime");   // TON
   #ResetVDComm := #SendToVDTimeOut.Q;
END_REGION

NETWORK
TITLE = **** 4.4 - Machine status - Calculated **** Init Done
// Init Done

      A     #I_PhoneAlarmReq1;
      O     #RequestCommand1;
      FP    #InitDoneEdge[1];
      =     #InitDone[1];

      A     #I_PhoneAlarmReq2;
      O     #RequestCommand2;
      FP    #InitDoneEdge[2];
      =     #InitDone[2];

      A     #I_PhoneAlarmReq3;
      O     #RequestCommand3;
      FP    #InitDoneEdge[3];
      =     #InitDone[3];

      A     #I_PhoneAlarmReq4;
      O     #RequestCommand4;
      FP    #InitDoneEdge[4];
      =     #InitDone[4];

      A     #I_PhoneAlarmReq5;
      O     #RequestCommand5;
      FP    #InitDoneEdge[5];
      =     #InitDone[5];

      A     #I_PhoneAlarmReq6;
      O     #RequestCommand6;
      FP    #InitDoneEdge[6];
      =     #InitDone[6];

      A     #I_PhoneAlarmReq7;
      O     #RequestCommand7;
      FP    #InitDoneEdge[7];
      =     #InitDone[7];

      A     #I_PhoneAlarmReq8;
      O     #RequestCommand8;
      FP    #InitDoneEdge[8];
      =     #InitDone[8];

      A     #I_PhoneAlarmReq9;
      O     #RequestCommand9;
      FP    #InitDoneEdge[9];
      =     #InitDone[9];

      A     #I_PhoneAlarmReq10;
      O     #RequestCommand10;
      FP    #InitDoneEdge[10];
      =     #InitDone[10];

      A     #I_PhoneAlarmReq11;
      O     #RequestCommand11;
      FP    #InitDoneEdge[11];
      =     #InitDone[11];

      A     #I_PhoneAlarmReq12;
      O     #RequestCommand12;
      FP    #InitDoneEdge[12];
      =     #InitDone[12];

      A     #I_PhoneAlarmReq13;
      O     #RequestCommand13;
      FP    #InitDoneEdge[13];
      =     #InitDone[13];

      A     #I_PhoneAlarmReq14;
      O     #RequestCommand14;
      FP    #InitDoneEdge[14];
      =     #InitDone[14];

      A     #I_PhoneAlarmReq15;
      O     #RequestCommand15;
      FP    #InitDoneEdge[15];
      =     #InitDone[15];

      A     #I_PhoneAlarmReq16;
      O     #RequestCommand16;
      FP    #InitDoneEdge[16];
      =     #InitDone[16];


REGION Network 8: **** 4.4 - Machine Status - Calculation **** Request PhoneAlarm Stn1 Filter
   // Filter
   #_Filter1(IN := #I_PhoneAlarmReq1, PT := #C_FilterMessage1, ET => "NotUsedTime");   // TON
   #PhoneAlarmReqActiveStn1 := #_Filter1.Q;
END_REGION

REGION Network 9: **** 4.4 - Machine Status - Calculation **** Request PhoneAlarm Stn1
   // Request PhoneAlarm Stn1
   IF #PhoneAlarmReqActiveStn1 OR #RequestCommand1 THEN
       #ReqPhoneAlarm[1] := TRUE;   // SR flip-flop
   END_IF;
   IF #Done[1] THEN #ReqPhoneAlarm[1] := FALSE; END_IF;
END_REGION

REGION Network 10: **** 4.4 - Machine Status - Calculation **** Request PhoneAlarm Stn2 Filter
   // Filter
   #_Filter2(IN := #I_PhoneAlarmReq2, PT := #C_FilterMessage2, ET => "NotUsedTime");   // TON
   #PhoneAlarmReqActiveStn2 := #_Filter2.Q;
END_REGION

REGION Network 11: **** 4.4 - Machine Status - Calculation **** Request PhoneAlarm Stn2
   // Request PhoneAlarm Stn2
   IF #PhoneAlarmReqActiveStn2 OR #RequestCommand2 THEN
       #ReqPhoneAlarm[2] := TRUE;   // SR flip-flop
   END_IF;
   IF #Done[2] THEN #ReqPhoneAlarm[2] := FALSE; END_IF;
END_REGION

REGION Network 12: **** 4.4 - Machine Status - Calculation **** Request PhoneAlarm Stn3 Filter
   // Filter
   #_Filter3(IN := #I_PhoneAlarmReq3, PT := #C_FilterMessage3, ET => "NotUsedTime");   // TON
   #PhoneAlarmReqActiveStn3 := #_Filter3.Q;
END_REGION

REGION Network 13: **** 4.4 - Machine Status - Calculation **** Request PhoneAlarm Stn3
   // Request PhoneAlarm Stn3
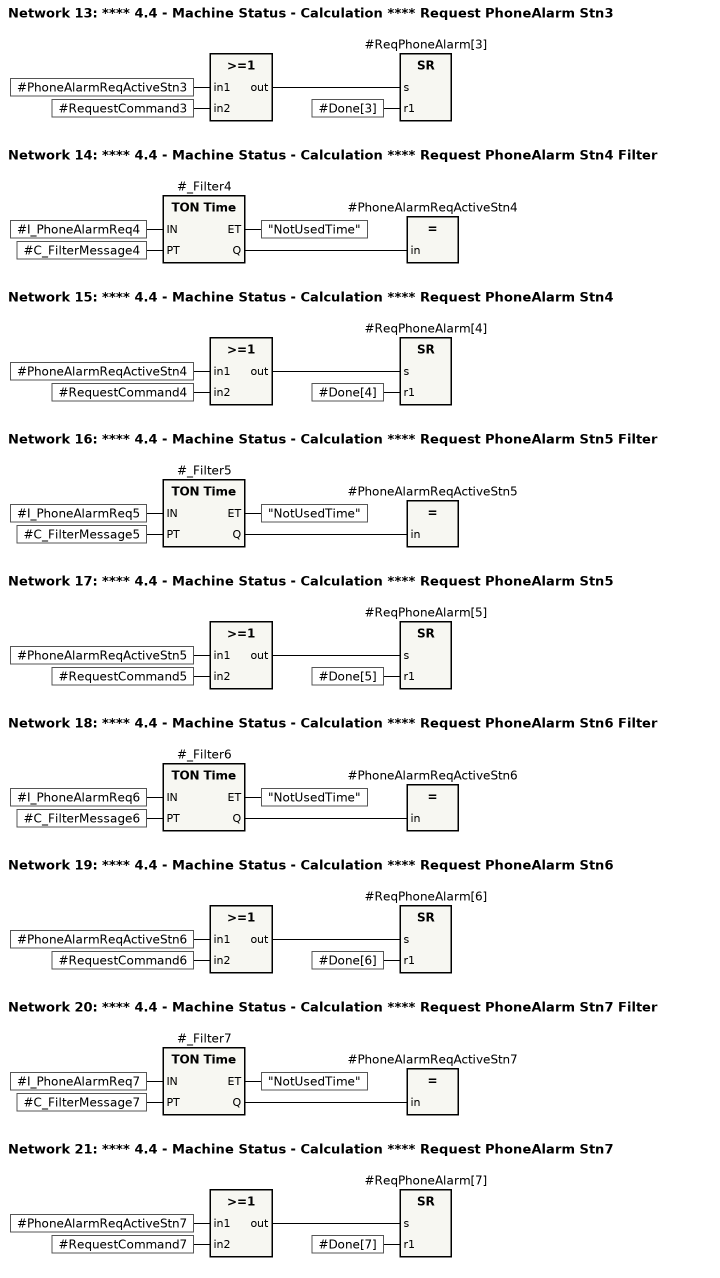
   IF #PhoneAlarmReqActiveStn3 OR #RequestCommand3 THEN
       #ReqPhoneAlarm[3] := TRUE;   // SR flip-flop
   END_IF;
   IF #Done[3] THEN #ReqPhoneAlarm[3] := FALSE; END_IF;
END_REGION

REGION Network 14: **** 4.4 - Machine Status - Calculation **** Request PhoneAlarm Stn4 Filter
   // Filter
   #_Filter4(IN := #I_PhoneAlarmReq4, PT := #C_FilterMessage4, ET => "NotUsedTime");   // TON
   #PhoneAlarmReqActiveStn4 := #_Filter4.Q;
END_REGION

REGION Network 15: **** 4.4 - Machine Status - Calculation **** Request PhoneAlarm Stn4
   // Request PhoneAlarm Stn4
   IF #PhoneAlarmReqActiveStn4 OR #RequestCommand4 THEN
       #ReqPhoneAlarm[4] := TRUE;   // SR flip-flop
   END_IF;
   IF #Done[4] THEN #ReqPhoneAlarm[4] := FALSE; END_IF;
END_REGION

REGION Network 16: **** 4.4 - Machine Status - Calculation **** Request PhoneAlarm Stn5 Filter
   // Filter
   #_Filter5(IN := #I_PhoneAlarmReq5, PT := #C_FilterMessage5, ET => "NotUsedTime");   // TON
   #PhoneAlarmReqActiveStn5 := #_Filter5.Q;
END_REGION

REGION Network 17: **** 4.4 - Machine Status - Calculation **** Request PhoneAlarm Stn5
   // Request PhoneAlarm Stn5
   IF #PhoneAlarmReqActiveStn5 OR #RequestCommand5 THEN
       #ReqPhoneAlarm[5] := TRUE;   // SR flip-flop
   END_IF;
   IF #Done[5] THEN #ReqPhoneAlarm[5] := FALSE; END_IF;
END_REGION

REGION Network 18: **** 4.4 - Machine Status - Calculation **** Request PhoneAlarm Stn6 Filter
   // Filter
   #_Filter6(IN := #I_PhoneAlarmReq6, PT := #C_FilterMessage6, ET => "NotUsedTime");   // TON
   #PhoneAlarmReqActiveStn6 := #_Filter6.Q;
END_REGION

REGION Network 19: **** 4.4 - Machine Status - Calculation **** Request PhoneAlarm Stn6
   // Request PhoneAlarm Stn6
   IF #PhoneAlarmReqActiveStn6 OR #RequestCommand6 THEN
       #ReqPhoneAlarm[6] := TRUE;   // SR flip-flop
   END_IF;
   IF #Done[6] THEN #ReqPhoneAlarm[6] := FALSE; END_IF;
END_REGION

REGION Network 20: **** 4.4 - Machine Status - Calculation **** Request PhoneAlarm Stn7 Filter
   // Filter
   #_Filter7(IN := #I_PhoneAlarmReq7, PT := #C_FilterMessage7, ET => "NotUsedTime");   // TON
   #PhoneAlarmReqActiveStn7 := #_Filter7.Q;
END_REGION

REGION Network 21: **** 4.4 - Machine Status - Calculation **** Request PhoneAlarm Stn7
   // Request PhoneAlarm Stn7
   IF #PhoneAlarmReqActiveStn7 OR #RequestCommand7 THEN
       #ReqPhoneAlarm[7] := TRUE;   // SR flip-flop
   END_IF;
   IF #Done[7] THEN #ReqPhoneAlarm[7] := FALSE; END_IF;
END_REGION

REGION Network 22: **** 4.4 - Machine Status - Calculation **** Request PhoneAlarm Stn8 Filter
   // Filter
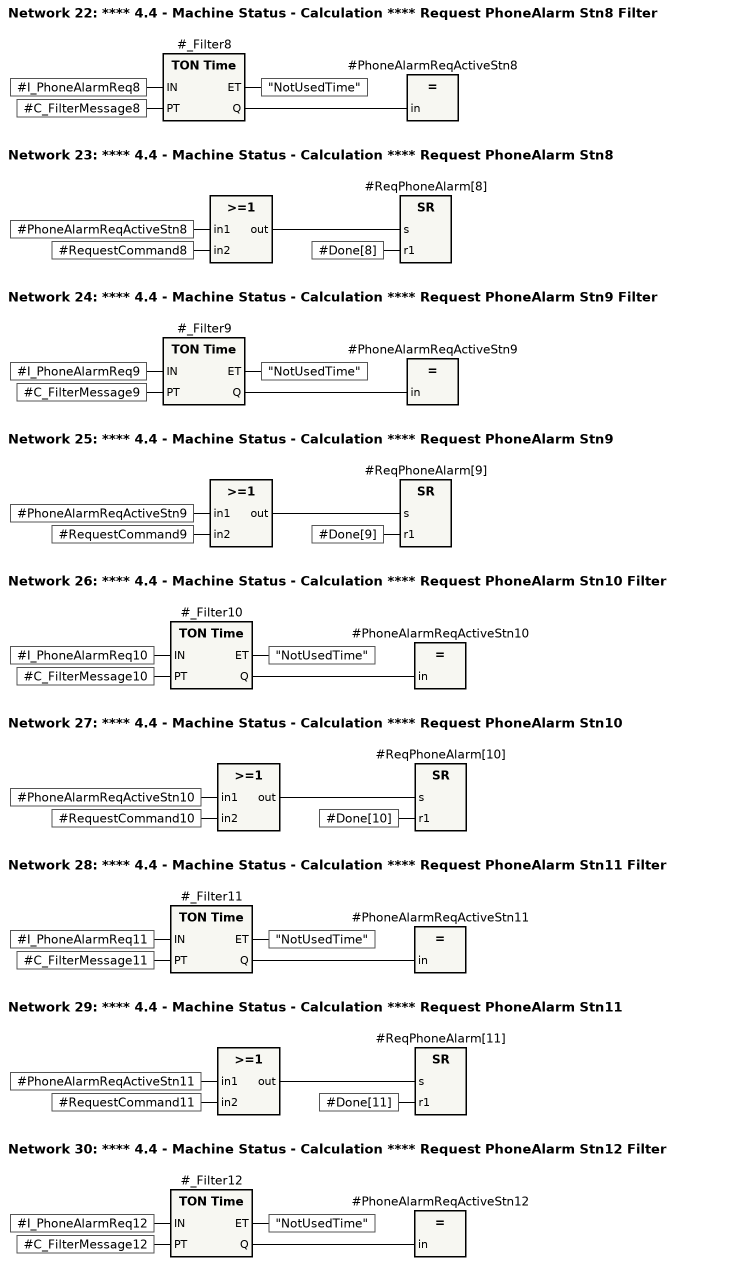
   #_Filter8(IN := #I_PhoneAlarmReq8, PT := #C_FilterMessage8, ET => "NotUsedTime");   // TON
   #PhoneAlarmReqActiveStn8 := #_Filter8.Q;
END_REGION

REGION Network 23: **** 4.4 - Machine Status - Calculation **** Request PhoneAlarm Stn8
   // Request PhoneAlarm Stn8
   IF #PhoneAlarmReqActiveStn8 OR #RequestCommand8 THEN
       #ReqPhoneAlarm[8] := TRUE;   // SR flip-flop
   END_IF;
   IF #Done[8] THEN #ReqPhoneAlarm[8] := FALSE; END_IF;
END_REGION

REGION Network 24: **** 4.4 - Machine Status - Calculation **** Request PhoneAlarm Stn9 Filter
   // Filter
   #_Filter9(IN := #I_PhoneAlarmReq9, PT := #C_FilterMessage9, ET => "NotUsedTime");   // TON
   #PhoneAlarmReqActiveStn9 := #_Filter9.Q;
END_REGION

REGION Network 25: **** 4.4 - Machine Status - Calculation **** Request PhoneAlarm Stn9
   // Request PhoneAlarm Stn9
   IF #PhoneAlarmReqActiveStn9 OR #RequestCommand9 THEN
       #ReqPhoneAlarm[9] := TRUE;   // SR flip-flop
   END_IF;
   IF #Done[9] THEN #ReqPhoneAlarm[9] := FALSE; END_IF;
END_REGION

REGION Network 26: **** 4.4 - Machine Status - Calculation **** Request PhoneAlarm Stn10 Filter
   // Filter
   #_Filter10(IN := #I_PhoneAlarmReq10, PT := #C_FilterMessage10, ET => "NotUsedTime");   // TON
   #PhoneAlarmReqActiveStn10 := #_Filter10.Q;
END_REGION

REGION Network 27: **** 4.4 - Machine Status - Calculation **** Request PhoneAlarm Stn10
   // Request PhoneAlarm Stn10
   IF #PhoneAlarmReqActiveStn10 OR #RequestCommand10 THEN
       #ReqPhoneAlarm[10] := TRUE;   // SR flip-flop
   END_IF;
   IF #Done[10] THEN #ReqPhoneAlarm[10] := FALSE; END_IF;
END_REGION

REGION Network 28: **** 4.4 - Machine Status - Calculation **** Request PhoneAlarm Stn11 Filter
   // Filter
   #_Filter11(IN := #I_PhoneAlarmReq11, PT := #C_FilterMessage11, ET => "NotUsedTime");   // TON
   #PhoneAlarmReqActiveStn11 := #_Filter11.Q;
END_REGION

REGION Network 29: **** 4.4 - Machine Status - Calculation **** Request PhoneAlarm Stn11
   // Request PhoneAlarm Stn11
   IF #PhoneAlarmReqActiveStn11 OR #RequestCommand11 THEN
       #ReqPhoneAlarm[11] := TRUE;   // SR flip-flop
   END_IF;
   IF #Done[11] THEN #ReqPhoneAlarm[11] := FALSE; END_IF;
END_REGION

REGION Network 30: **** 4.4 - Machine Status - Calculation **** Request PhoneAlarm Stn12 Filter
   // Filter
   #_Filter12(IN := #I_PhoneAlarmReq12, PT := #C_FilterMessage12, ET => "NotUsedTime");   // TON
   #PhoneAlarmReqActiveStn12 := #_Filter12.Q;
END_REGION

REGION Network 31: **** 4.4 - Machine Status - Calculation **** Request PhoneAlarm Stn12
   // Request PhoneAlarm Stn12
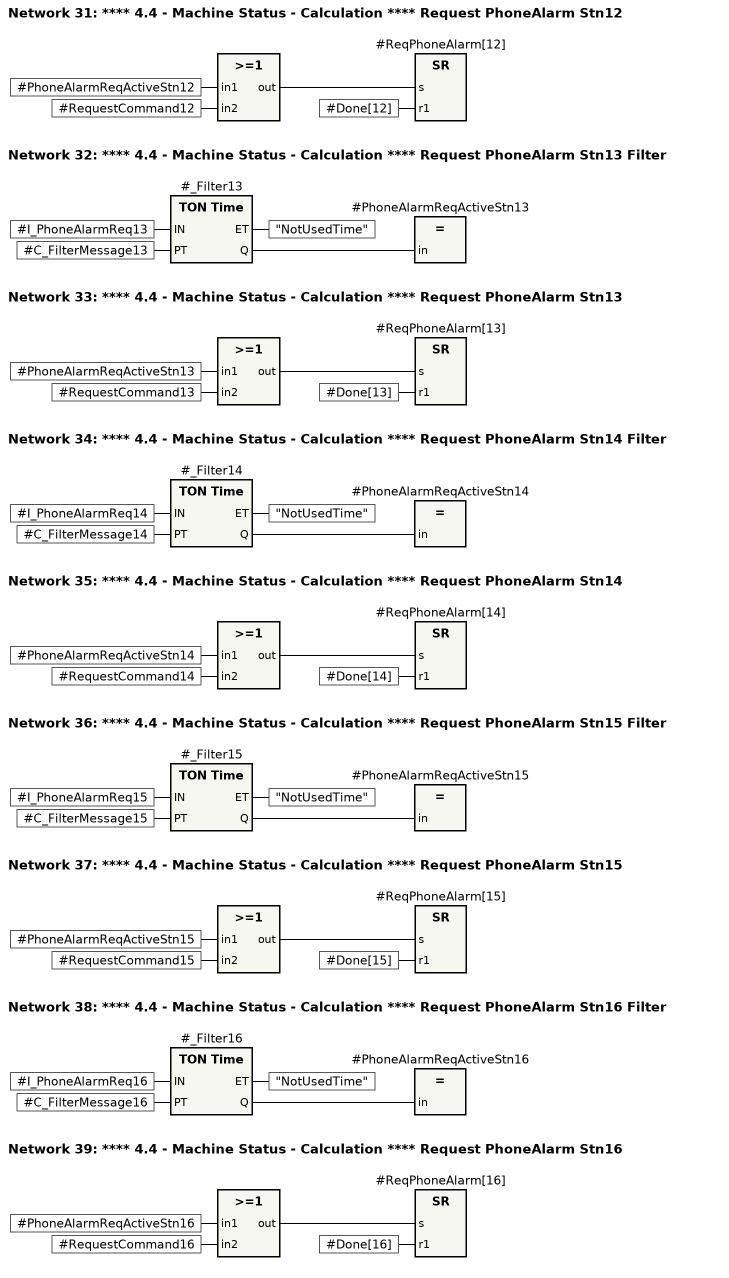
   IF #PhoneAlarmReqActiveStn12 OR #RequestCommand12 THEN
       #ReqPhoneAlarm[12] := TRUE;   // SR flip-flop
   END_IF;
   IF #Done[12] THEN #ReqPhoneAlarm[12] := FALSE; END_IF;
END_REGION

REGION Network 32: **** 4.4 - Machine Status - Calculation **** Request PhoneAlarm Stn13 Filter
   // Filter
   #_Filter13(IN := #I_PhoneAlarmReq13, PT := #C_FilterMessage13, ET => "NotUsedTime");   // TON
   #PhoneAlarmReqActiveStn13 := #_Filter13.Q;
END_REGION

REGION Network 33: **** 4.4 - Machine Status - Calculation **** Request PhoneAlarm Stn13
   // Request PhoneAlarm Stn13
   IF #PhoneAlarmReqActiveStn13 OR #RequestCommand13 THEN
       #ReqPhoneAlarm[13] := TRUE;   // SR flip-flop
   END_IF;
   IF #Done[13] THEN #ReqPhoneAlarm[13] := FALSE; END_IF;
END_REGION

REGION Network 34: **** 4.4 - Machine Status - Calculation **** Request PhoneAlarm Stn14 Filter
   // Filter
   #_Filter14(IN := #I_PhoneAlarmReq14, PT := #C_FilterMessage14, ET => "NotUsedTime");   // TON
   #PhoneAlarmReqActiveStn14 := #_Filter14.Q;
END_REGION

REGION Network 35: **** 4.4 - Machine Status - Calculation **** Request PhoneAlarm Stn14
   // Request PhoneAlarm Stn14
   IF #PhoneAlarmReqActiveStn14 OR #RequestCommand14 THEN
       #ReqPhoneAlarm[14] := TRUE;   // SR flip-flop
   END_IF;
   IF #Done[14] THEN #ReqPhoneAlarm[14] := FALSE; END_IF;
END_REGION

REGION Network 36: **** 4.4 - Machine Status - Calculation **** Request PhoneAlarm Stn15 Filter
   // Filter
   #_Filter15(IN := #I_PhoneAlarmReq15, PT := #C_FilterMessage15, ET => "NotUsedTime");   // TON
   #PhoneAlarmReqActiveStn15 := #_Filter15.Q;
END_REGION

REGION Network 37: **** 4.4 - Machine Status - Calculation **** Request PhoneAlarm Stn15
   // Request PhoneAlarm Stn15
   IF #PhoneAlarmReqActiveStn15 OR #RequestCommand15 THEN
       #ReqPhoneAlarm[15] := TRUE;   // SR flip-flop
   END_IF;
   IF #Done[15] THEN #ReqPhoneAlarm[15] := FALSE; END_IF;
END_REGION

REGION Network 38: **** 4.4 - Machine Status - Calculation **** Request PhoneAlarm Stn16 Filter
   // Filter
   #_Filter16(IN := #I_PhoneAlarmReq16, PT := #C_FilterMessage16, ET => "NotUsedTime");   // TON
   #PhoneAlarmReqActiveStn16 := #_Filter16.Q;
END_REGION

REGION Network 39: **** 4.4 - Machine Status - Calculation **** Request PhoneAlarm Stn16
   // Request PhoneAlarm Stn16
   IF #PhoneAlarmReqActiveStn16 OR #RequestCommand16 THEN
       #ReqPhoneAlarm[16] := TRUE;   // SR flip-flop
   END_IF;
   IF #Done[16] THEN #ReqPhoneAlarm[16] := FALSE; END_IF;
END_REGION

REGION Network 40: **** 4.4 - Machine Status - Calculation **** Message Request Done
   // Message Request Done
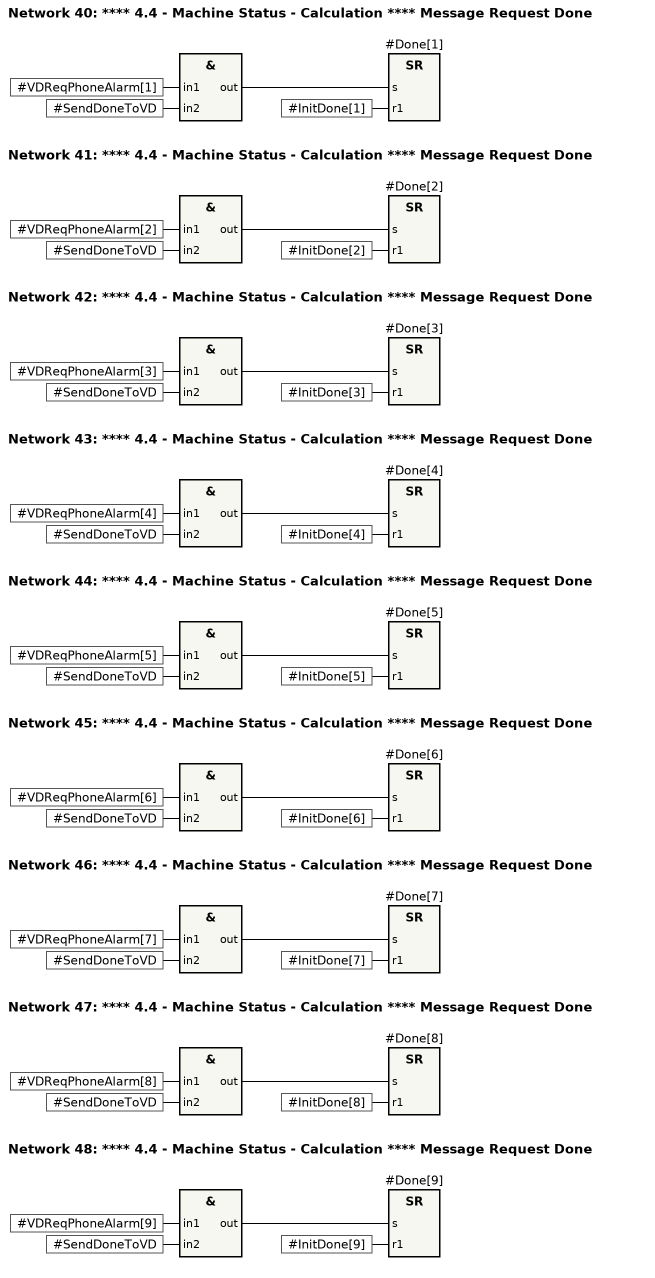
   IF #VDReqPhoneAlarm[1] AND #SendDoneToVD THEN
       #Done[1] := TRUE;   // SR flip-flop
   END_IF;
   IF #InitDone[1] THEN #Done[1] := FALSE; END_IF;
END_REGION

REGION Network 41: **** 4.4 - Machine Status - Calculation **** Message Request Done
   // Message Request Done
   IF #VDReqPhoneAlarm[2] AND #SendDoneToVD THEN
       #Done[2] := TRUE;   // SR flip-flop
   END_IF;
   IF #InitDone[2] THEN #Done[2] := FALSE; END_IF;
END_REGION

REGION Network 42: **** 4.4 - Machine Status - Calculation **** Message Request Done
   // Message Request Done
   IF #VDReqPhoneAlarm[3] AND #SendDoneToVD THEN
       #Done[3] := TRUE;   // SR flip-flop
   END_IF;
   IF #InitDone[3] THEN #Done[3] := FALSE; END_IF;
END_REGION

REGION Network 43: **** 4.4 - Machine Status - Calculation **** Message Request Done
   // Message Request Done
   IF #VDReqPhoneAlarm[4] AND #SendDoneToVD THEN
       #Done[4] := TRUE;   // SR flip-flop
   END_IF;
   IF #InitDone[4] THEN #Done[4] := FALSE; END_IF;
END_REGION

REGION Network 44: **** 4.4 - Machine Status - Calculation **** Message Request Done
   // Message Request Done
   IF #VDReqPhoneAlarm[5] AND #SendDoneToVD THEN
       #Done[5] := TRUE;   // SR flip-flop
   END_IF;
   IF #InitDone[5] THEN #Done[5] := FALSE; END_IF;
END_REGION

REGION Network 45: **** 4.4 - Machine Status - Calculation **** Message Request Done
   // Message Request Done
   IF #VDReqPhoneAlarm[6] AND #SendDoneToVD THEN
       #Done[6] := TRUE;   // SR flip-flop
   END_IF;
   IF #InitDone[6] THEN #Done[6] := FALSE; END_IF;
END_REGION

REGION Network 46: **** 4.4 - Machine Status - Calculation **** Message Request Done
   // Message Request Done
   IF #VDReqPhoneAlarm[7] AND #SendDoneToVD THEN
       #Done[7] := TRUE;   // SR flip-flop
   END_IF;
   IF #InitDone[7] THEN #Done[7] := FALSE; END_IF;
END_REGION

REGION Network 47: **** 4.4 - Machine Status - Calculation **** Message Request Done
   // Message Request Done
   IF #VDReqPhoneAlarm[8] AND #SendDoneToVD THEN
       #Done[8] := TRUE;   // SR flip-flop
   END_IF;
   IF #InitDone[8] THEN #Done[8] := FALSE; END_IF;
END_REGION

REGION Network 48: **** 4.4 - Machine Status - Calculation **** Message Request Done
   // Message Request Done
   IF #VDReqPhoneAlarm[9] AND #SendDoneToVD THEN
       #Done[9] := TRUE;   // SR flip-flop
   END_IF;
   IF #InitDone[9] THEN #Done[9] := FALSE; END_IF;
END_REGION

REGION Network 49: **** 4.4 - Machine Status - Calculation **** Message Request Done
   // Message Request Done
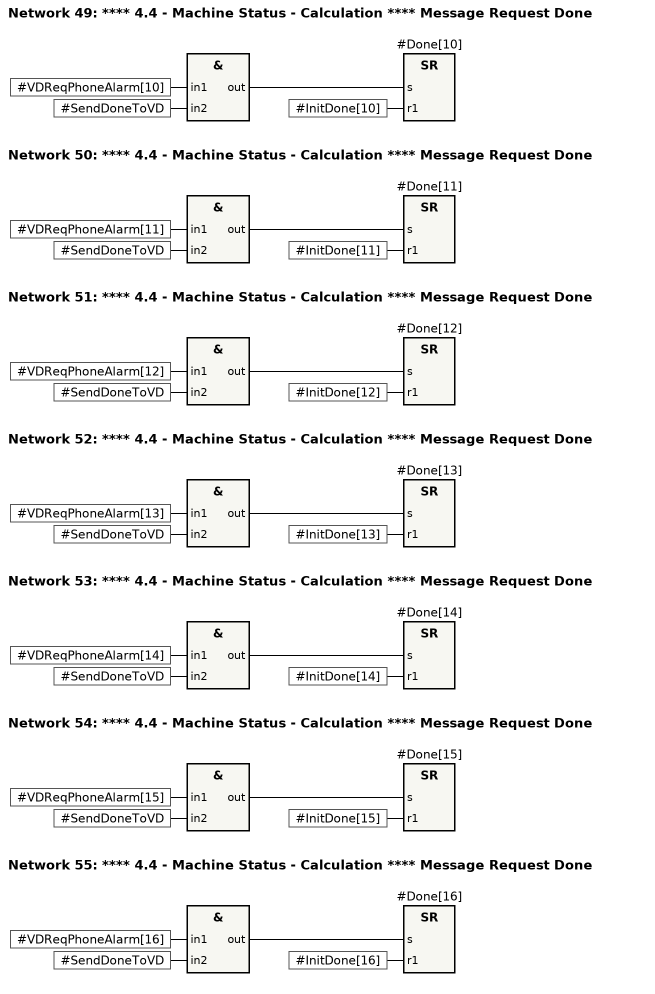
   IF #VDReqPhoneAlarm[10] AND #SendDoneToVD THEN
       #Done[10] := TRUE;   // SR flip-flop
   END_IF;
   IF #InitDone[10] THEN #Done[10] := FALSE; END_IF;
END_REGION

REGION Network 50: **** 4.4 - Machine Status - Calculation **** Message Request Done
   // Message Request Done
   IF #VDReqPhoneAlarm[11] AND #SendDoneToVD THEN
       #Done[11] := TRUE;   // SR flip-flop
   END_IF;
   IF #InitDone[11] THEN #Done[11] := FALSE; END_IF;
END_REGION

REGION Network 51: **** 4.4 - Machine Status - Calculation **** Message Request Done
   // Message Request Done
   IF #VDReqPhoneAlarm[12] AND #SendDoneToVD THEN
       #Done[12] := TRUE;   // SR flip-flop
   END_IF;
   IF #InitDone[12] THEN #Done[12] := FALSE; END_IF;
END_REGION

REGION Network 52: **** 4.4 - Machine Status - Calculation **** Message Request Done
   // Message Request Done
   IF #VDReqPhoneAlarm[13] AND #SendDoneToVD THEN
       #Done[13] := TRUE;   // SR flip-flop
   END_IF;
   IF #InitDone[13] THEN #Done[13] := FALSE; END_IF;
END_REGION

REGION Network 53: **** 4.4 - Machine Status - Calculation **** Message Request Done
   // Message Request Done
   IF #VDReqPhoneAlarm[14] AND #SendDoneToVD THEN
       #Done[14] := TRUE;   // SR flip-flop
   END_IF;
   IF #InitDone[14] THEN #Done[14] := FALSE; END_IF;
END_REGION

REGION Network 54: **** 4.4 - Machine Status - Calculation **** Message Request Done
   // Message Request Done
   IF #VDReqPhoneAlarm[15] AND #SendDoneToVD THEN
       #Done[15] := TRUE;   // SR flip-flop
   END_IF;
   IF #InitDone[15] THEN #Done[15] := FALSE; END_IF;
END_REGION

REGION Network 55: **** 4.4 - Machine Status - Calculation **** Message Request Done
   // Message Request Done
   IF #VDReqPhoneAlarm[16] AND #SendDoneToVD THEN
       #Done[16] := TRUE;   // SR flip-flop
   END_IF;
   IF #InitDone[16] THEN #Done[16] := FALSE; END_IF;
END_REGION

REGION Network 56: **** 4.4 - Machine Status - Calculation **** Que Message Request 1 / **** 4.4 - Machine Status - Calculation **** Queue Message Request 1
   // Que Message Request 1 / Queue Message Request 1
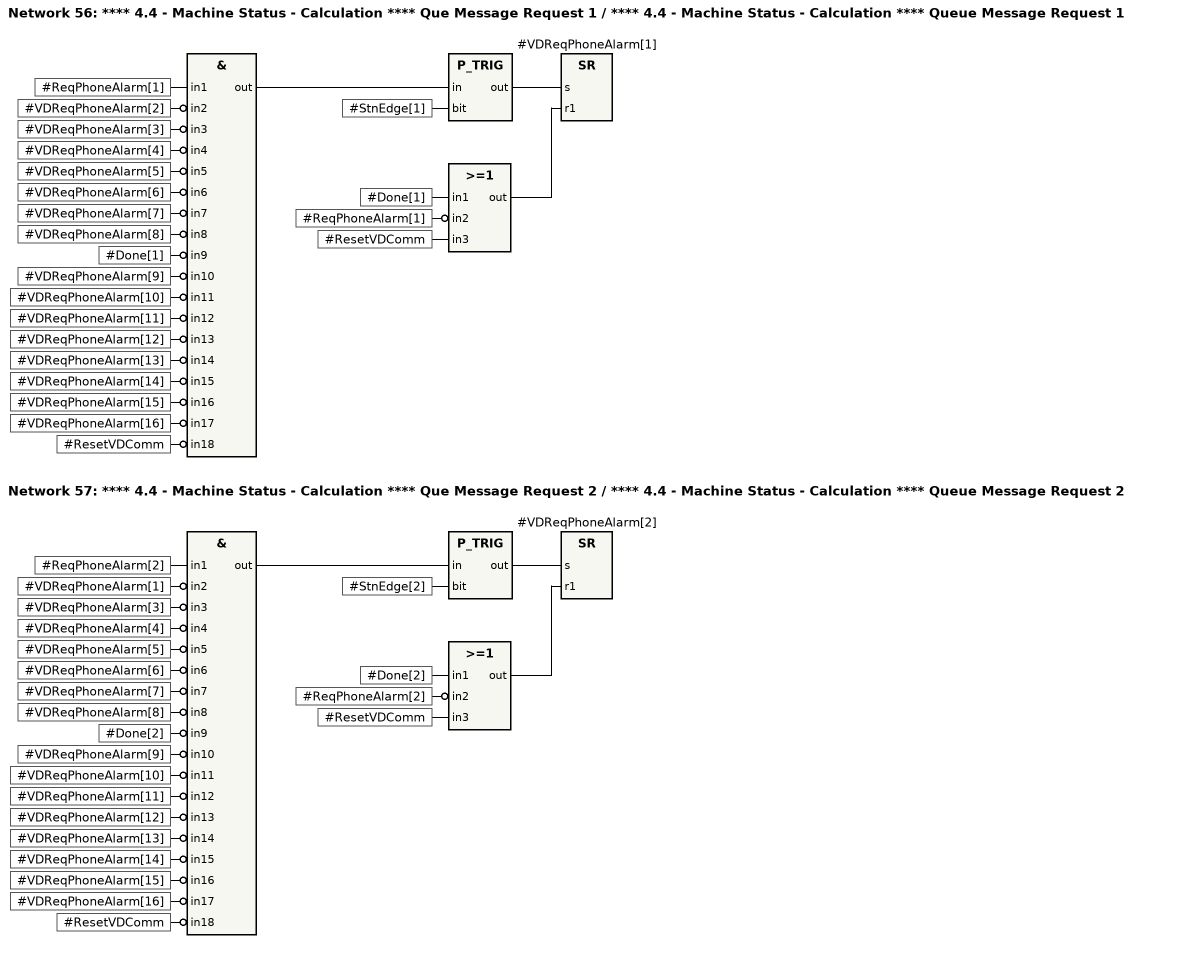
   #_w1 := #ReqPhoneAlarm[1] AND NOT #VDReqPhoneAlarm[2] AND NOT #VDReqPhoneAlarm[3] AND NOT #VDReqPhoneAlarm[4] AND NOT #VDReqPhoneAlarm[5] AND NOT #VDReqPhoneAlarm[6] AND NOT #VDReqPhoneAlarm[7] AND NOT #VDReqPhoneAlarm[8] AND NOT #Done[1] AND NOT #VDReqPhoneAlarm[9] AND NOT #VDReqPhoneAlarm[10] AND NOT #VDReqPhoneAlarm[11] AND NOT #VDReqPhoneAlarm[12] AND NOT #VDReqPhoneAlarm[13] AND NOT #VDReqPhoneAlarm[14] AND NOT #VDReqPhoneAlarm[15] AND NOT #VDReqPhoneAlarm[16] AND NOT #ResetVDComm;
   #_w2 := #_w1 AND NOT #StnEdge[1];   // rising edge
   #StnEdge[1] := #_w1;
   IF #_w2 THEN
       #VDReqPhoneAlarm[1] := TRUE;   // SR flip-flop
   END_IF;
   IF #Done[1] OR NOT #ReqPhoneAlarm[1] OR #ResetVDComm THEN #VDReqPhoneAlarm[1] := FALSE; END_IF;
END_REGION

REGION Network 57: **** 4.4 - Machine Status - Calculation **** Que Message Request 2 / **** 4.4 - Machine Status - Calculation **** Queue Message Request 2
   // Que Message Request 2 / Queue Message Request 2
   #_w1 := #ReqPhoneAlarm[2] AND NOT #VDReqPhoneAlarm[1] AND NOT #VDReqPhoneAlarm[3] AND NOT #VDReqPhoneAlarm[4] AND NOT #VDReqPhoneAlarm[5] AND NOT #VDReqPhoneAlarm[6] AND NOT #VDReqPhoneAlarm[7] AND NOT #VDReqPhoneAlarm[8] AND NOT #Done[2] AND NOT #VDReqPhoneAlarm[9] AND NOT #VDReqPhoneAlarm[10] AND NOT #VDReqPhoneAlarm[11] AND NOT #VDReqPhoneAlarm[12] AND NOT #VDReqPhoneAlarm[13] AND NOT #VDReqPhoneAlarm[14] AND NOT #VDReqPhoneAlarm[15] AND NOT #VDReqPhoneAlarm[16] AND NOT #ResetVDComm;
   #_w2 := #_w1 AND NOT #StnEdge[2];   // rising edge
   #StnEdge[2] := #_w1;
   IF #_w2 THEN
       #VDReqPhoneAlarm[2] := TRUE;   // SR flip-flop
   END_IF;
   IF #Done[2] OR NOT #ReqPhoneAlarm[2] OR #ResetVDComm THEN #VDReqPhoneAlarm[2] := FALSE; END_IF;
END_REGION

REGION Network 58: **** 4.4 - Machine Status - Calculation **** Que Message Request 3 / **** 4.4 - Machine Status - Calculation **** Queue Message Request 3
   // Que Message Request 3 / Queue Message Request 3
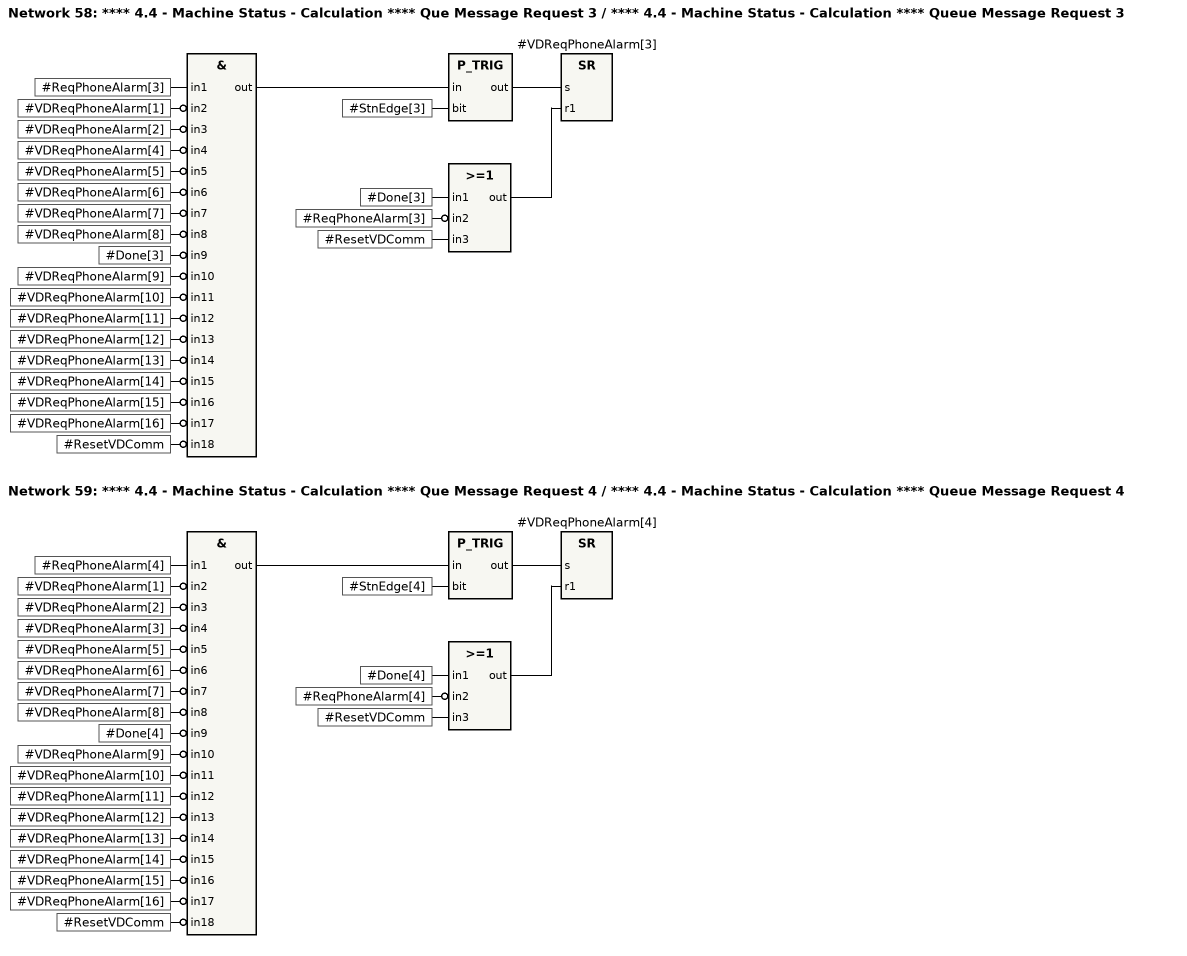
   #_w1 := #ReqPhoneAlarm[3] AND NOT #VDReqPhoneAlarm[1] AND NOT #VDReqPhoneAlarm[2] AND NOT #VDReqPhoneAlarm[4] AND NOT #VDReqPhoneAlarm[5] AND NOT #VDReqPhoneAlarm[6] AND NOT #VDReqPhoneAlarm[7] AND NOT #VDReqPhoneAlarm[8] AND NOT #Done[3] AND NOT #VDReqPhoneAlarm[9] AND NOT #VDReqPhoneAlarm[10] AND NOT #VDReqPhoneAlarm[11] AND NOT #VDReqPhoneAlarm[12] AND NOT #VDReqPhoneAlarm[13] AND NOT #VDReqPhoneAlarm[14] AND NOT #VDReqPhoneAlarm[15] AND NOT #VDReqPhoneAlarm[16] AND NOT #ResetVDComm;
   #_w2 := #_w1 AND NOT #StnEdge[3];   // rising edge
   #StnEdge[3] := #_w1;
   IF #_w2 THEN
       #VDReqPhoneAlarm[3] := TRUE;   // SR flip-flop
   END_IF;
   IF #Done[3] OR NOT #ReqPhoneAlarm[3] OR #ResetVDComm THEN #VDReqPhoneAlarm[3] := FALSE; END_IF;
END_REGION

REGION Network 59: **** 4.4 - Machine Status - Calculation **** Que Message Request 4 / **** 4.4 - Machine Status - Calculation **** Queue Message Request 4
   // Que Message Request 4 / Queue Message Request 4
   #_w1 := #ReqPhoneAlarm[4] AND NOT #VDReqPhoneAlarm[1] AND NOT #VDReqPhoneAlarm[2] AND NOT #VDReqPhoneAlarm[3] AND NOT #VDReqPhoneAlarm[5] AND NOT #VDReqPhoneAlarm[6] AND NOT #VDReqPhoneAlarm[7] AND NOT #VDReqPhoneAlarm[8] AND NOT #Done[4] AND NOT #VDReqPhoneAlarm[9] AND NOT #VDReqPhoneAlarm[10] AND NOT #VDReqPhoneAlarm[11] AND NOT #VDReqPhoneAlarm[12] AND NOT #VDReqPhoneAlarm[13] AND NOT #VDReqPhoneAlarm[14] AND NOT #VDReqPhoneAlarm[15] AND NOT #VDReqPhoneAlarm[16] AND NOT #ResetVDComm;
   #_w2 := #_w1 AND NOT #StnEdge[4];   // rising edge
   #StnEdge[4] := #_w1;
   IF #_w2 THEN
       #VDReqPhoneAlarm[4] := TRUE;   // SR flip-flop
   END_IF;
   IF #Done[4] OR NOT #ReqPhoneAlarm[4] OR #ResetVDComm THEN #VDReqPhoneAlarm[4] := FALSE; END_IF;
END_REGION

REGION Network 60: **** 4.4 - Machine Status - Calculation **** Que Message Request 5 / **** 4.4 - Machine Status - Calculation **** Queue Message Request 5
   // Que Message Request 5 / Queue Message Request 5
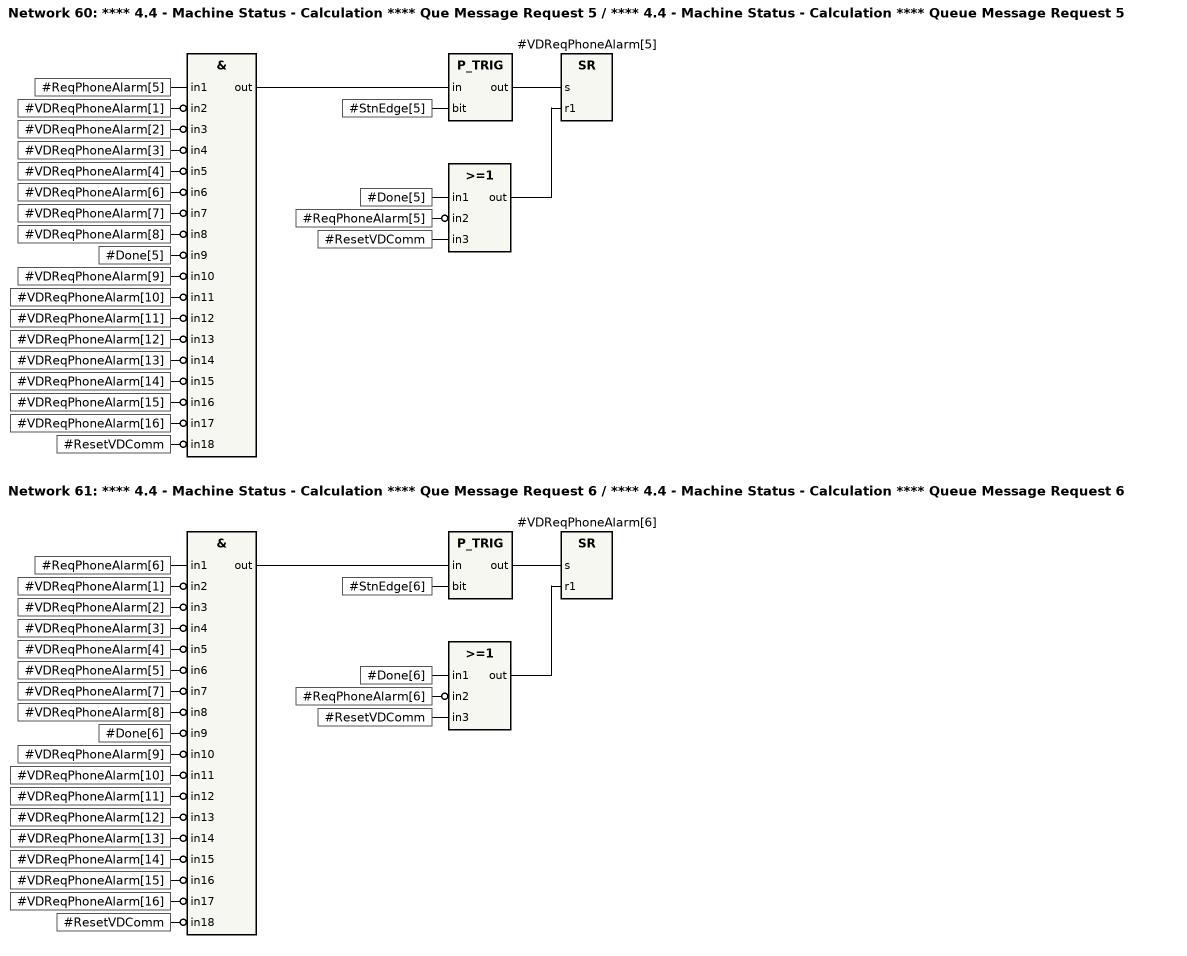
   #_w1 := #ReqPhoneAlarm[5] AND NOT #VDReqPhoneAlarm[1] AND NOT #VDReqPhoneAlarm[2] AND NOT #VDReqPhoneAlarm[3] AND NOT #VDReqPhoneAlarm[4] AND NOT #VDReqPhoneAlarm[6] AND NOT #VDReqPhoneAlarm[7] AND NOT #VDReqPhoneAlarm[8] AND NOT #Done[5] AND NOT #VDReqPhoneAlarm[9] AND NOT #VDReqPhoneAlarm[10] AND NOT #VDReqPhoneAlarm[11] AND NOT #VDReqPhoneAlarm[12] AND NOT #VDReqPhoneAlarm[13] AND NOT #VDReqPhoneAlarm[14] AND NOT #VDReqPhoneAlarm[15] AND NOT #VDReqPhoneAlarm[16] AND NOT #ResetVDComm;
   #_w2 := #_w1 AND NOT #StnEdge[5];   // rising edge
   #StnEdge[5] := #_w1;
   IF #_w2 THEN
       #VDReqPhoneAlarm[5] := TRUE;   // SR flip-flop
   END_IF;
   IF #Done[5] OR NOT #ReqPhoneAlarm[5] OR #ResetVDComm THEN #VDReqPhoneAlarm[5] := FALSE; END_IF;
END_REGION

REGION Network 61: **** 4.4 - Machine Status - Calculation **** Que Message Request 6 / **** 4.4 - Machine Status - Calculation **** Queue Message Request 6
   // Que Message Request 6 / Queue Message Request 6
   #_w1 := #ReqPhoneAlarm[6] AND NOT #VDReqPhoneAlarm[1] AND NOT #VDReqPhoneAlarm[2] AND NOT #VDReqPhoneAlarm[3] AND NOT #VDReqPhoneAlarm[4] AND NOT #VDReqPhoneAlarm[5] AND NOT #VDReqPhoneAlarm[7] AND NOT #VDReqPhoneAlarm[8] AND NOT #Done[6] AND NOT #VDReqPhoneAlarm[9] AND NOT #VDReqPhoneAlarm[10] AND NOT #VDReqPhoneAlarm[11] AND NOT #VDReqPhoneAlarm[12] AND NOT #VDReqPhoneAlarm[13] AND NOT #VDReqPhoneAlarm[14] AND NOT #VDReqPhoneAlarm[15] AND NOT #VDReqPhoneAlarm[16] AND NOT #ResetVDComm;
   #_w2 := #_w1 AND NOT #StnEdge[6];   // rising edge
   #StnEdge[6] := #_w1;
   IF #_w2 THEN
       #VDReqPhoneAlarm[6] := TRUE;   // SR flip-flop
   END_IF;
   IF #Done[6] OR NOT #ReqPhoneAlarm[6] OR #ResetVDComm THEN #VDReqPhoneAlarm[6] := FALSE; END_IF;
END_REGION

REGION Network 62: **** 4.4 - Machine Status - Calculation **** Que Message Request 7 / **** 4.4 - Machine Status - Calculation **** Queue Message Request 7
   // Que Message Request 7 / Queue Message Request 7
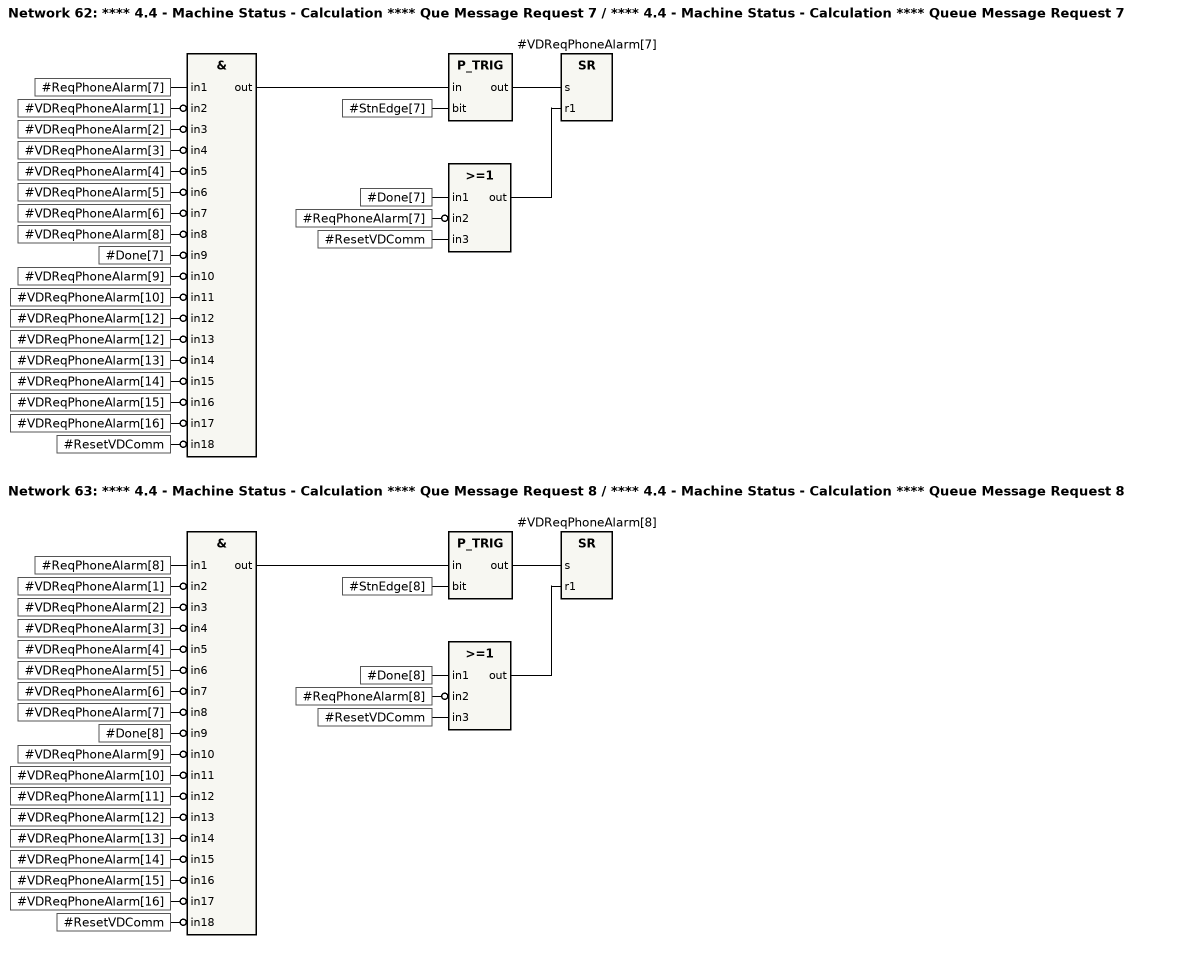
   #_w1 := #ReqPhoneAlarm[7] AND NOT #VDReqPhoneAlarm[1] AND NOT #VDReqPhoneAlarm[2] AND NOT #VDReqPhoneAlarm[3] AND NOT #VDReqPhoneAlarm[4] AND NOT #VDReqPhoneAlarm[5] AND NOT #VDReqPhoneAlarm[6] AND NOT #VDReqPhoneAlarm[8] AND NOT #Done[7] AND NOT #VDReqPhoneAlarm[9] AND NOT #VDReqPhoneAlarm[10] AND NOT #VDReqPhoneAlarm[12] AND NOT #VDReqPhoneAlarm[12] AND NOT #VDReqPhoneAlarm[13] AND NOT #VDReqPhoneAlarm[14] AND NOT #VDReqPhoneAlarm[15] AND NOT #VDReqPhoneAlarm[16] AND NOT #ResetVDComm;
   #_w2 := #_w1 AND NOT #StnEdge[7];   // rising edge
   #StnEdge[7] := #_w1;
   IF #_w2 THEN
       #VDReqPhoneAlarm[7] := TRUE;   // SR flip-flop
   END_IF;
   IF #Done[7] OR NOT #ReqPhoneAlarm[7] OR #ResetVDComm THEN #VDReqPhoneAlarm[7] := FALSE; END_IF;
END_REGION

REGION Network 63: **** 4.4 - Machine Status - Calculation **** Que Message Request 8 / **** 4.4 - Machine Status - Calculation **** Queue Message Request 8
   // Que Message Request 8 / Queue Message Request 8
   #_w1 := #ReqPhoneAlarm[8] AND NOT #VDReqPhoneAlarm[1] AND NOT #VDReqPhoneAlarm[2] AND NOT #VDReqPhoneAlarm[3] AND NOT #VDReqPhoneAlarm[4] AND NOT #VDReqPhoneAlarm[5] AND NOT #VDReqPhoneAlarm[6] AND NOT #VDReqPhoneAlarm[7] AND NOT #Done[8] AND NOT #VDReqPhoneAlarm[9] AND NOT #VDReqPhoneAlarm[10] AND NOT #VDReqPhoneAlarm[11] AND NOT #VDReqPhoneAlarm[12] AND NOT #VDReqPhoneAlarm[13] AND NOT #VDReqPhoneAlarm[14] AND NOT #VDReqPhoneAlarm[15] AND NOT #VDReqPhoneAlarm[16] AND NOT #ResetVDComm;
   #_w2 := #_w1 AND NOT #StnEdge[8];   // rising edge
   #StnEdge[8] := #_w1;
   IF #_w2 THEN
       #VDReqPhoneAlarm[8] := TRUE;   // SR flip-flop
   END_IF;
   IF #Done[8] OR NOT #ReqPhoneAlarm[8] OR #ResetVDComm THEN #VDReqPhoneAlarm[8] := FALSE; END_IF;
END_REGION

REGION Network 64: **** 4.4 - Machine Status - Calculation **** Que Message Request 9 / **** 4.4 - Machine Status - Calculation **** Queue Message Request 9
   // Que Message Request 9 / Queue Message Request 9
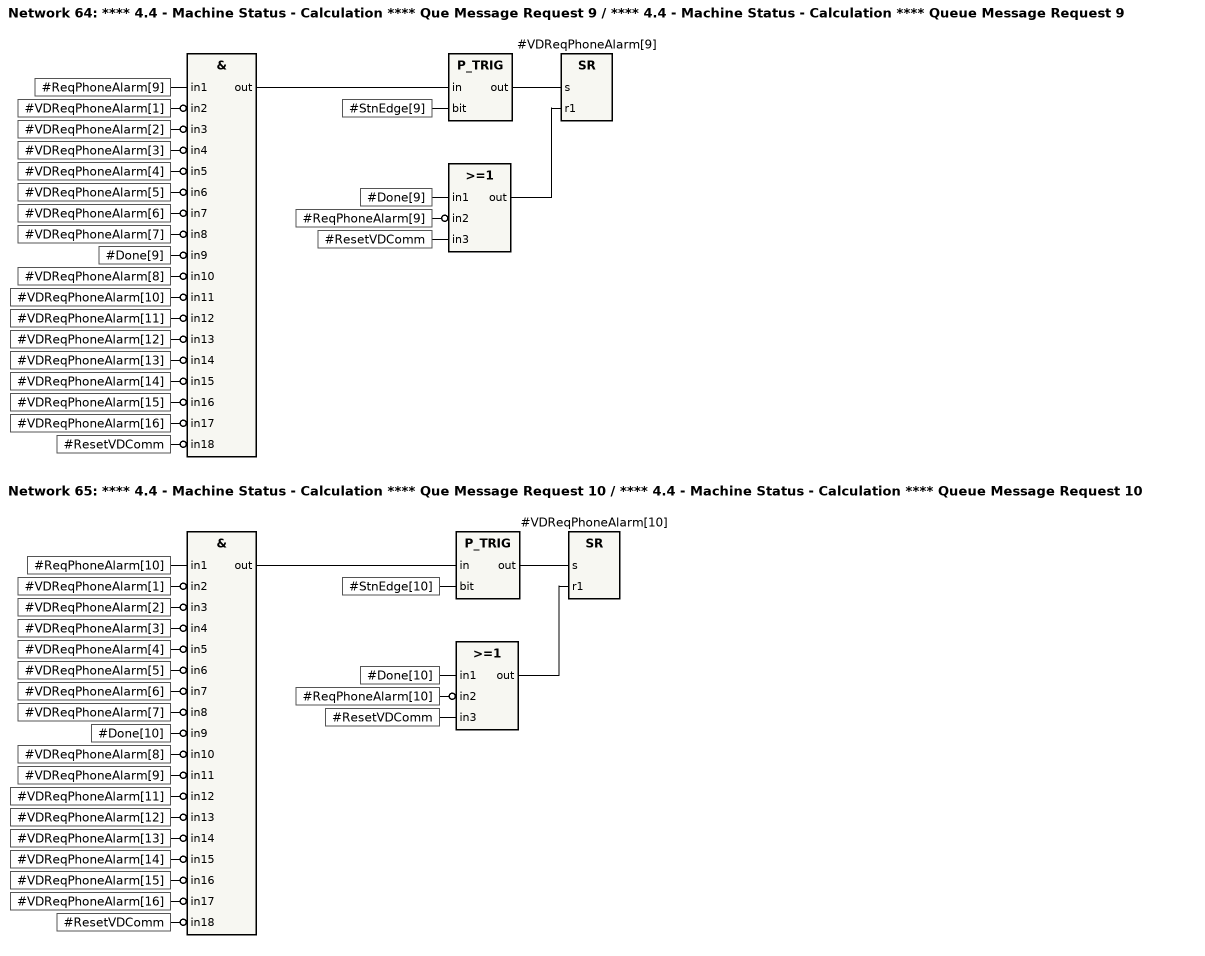
   #_w1 := #ReqPhoneAlarm[9] AND NOT #VDReqPhoneAlarm[1] AND NOT #VDReqPhoneAlarm[2] AND NOT #VDReqPhoneAlarm[3] AND NOT #VDReqPhoneAlarm[4] AND NOT #VDReqPhoneAlarm[5] AND NOT #VDReqPhoneAlarm[6] AND NOT #VDReqPhoneAlarm[7] AND NOT #Done[9] AND NOT #VDReqPhoneAlarm[8] AND NOT #VDReqPhoneAlarm[10] AND NOT #VDReqPhoneAlarm[11] AND NOT #VDReqPhoneAlarm[12] AND NOT #VDReqPhoneAlarm[13] AND NOT #VDReqPhoneAlarm[14] AND NOT #VDReqPhoneAlarm[15] AND NOT #VDReqPhoneAlarm[16] AND NOT #ResetVDComm;
   #_w2 := #_w1 AND NOT #StnEdge[9];   // rising edge
   #StnEdge[9] := #_w1;
   IF #_w2 THEN
       #VDReqPhoneAlarm[9] := TRUE;   // SR flip-flop
   END_IF;
   IF #Done[9] OR NOT #ReqPhoneAlarm[9] OR #ResetVDComm THEN #VDReqPhoneAlarm[9] := FALSE; END_IF;
END_REGION

REGION Network 65: **** 4.4 - Machine Status - Calculation **** Que Message Request 10 / **** 4.4 - Machine Status - Calculation **** Queue Message Request 10
   // Que Message Request 10 / Queue Message Request 10
   #_w1 := #ReqPhoneAlarm[10] AND NOT #VDReqPhoneAlarm[1] AND NOT #VDReqPhoneAlarm[2] AND NOT #VDReqPhoneAlarm[3] AND NOT #VDReqPhoneAlarm[4] AND NOT #VDReqPhoneAlarm[5] AND NOT #VDReqPhoneAlarm[6] AND NOT #VDReqPhoneAlarm[7] AND NOT #Done[10] AND NOT #VDReqPhoneAlarm[8] AND NOT #VDReqPhoneAlarm[9] AND NOT #VDReqPhoneAlarm[11] AND NOT #VDReqPhoneAlarm[12] AND NOT #VDReqPhoneAlarm[13] AND NOT #VDReqPhoneAlarm[14] AND NOT #VDReqPhoneAlarm[15] AND NOT #VDReqPhoneAlarm[16] AND NOT #ResetVDComm;
   #_w2 := #_w1 AND NOT #StnEdge[10];   // rising edge
   #StnEdge[10] := #_w1;
   IF #_w2 THEN
       #VDReqPhoneAlarm[10] := TRUE;   // SR flip-flop
   END_IF;
   IF #Done[10] OR NOT #ReqPhoneAlarm[10] OR #ResetVDComm THEN #VDReqPhoneAlarm[10] := FALSE; END_IF;
END_REGION

REGION Network 66: **** 4.4 - Machine Status - Calculation **** Que Message Request 11 / **** 4.4 - Machine Status - Calculation **** Queue Message Request 11
   // Que Message Request 11 / Queue Message Request 11
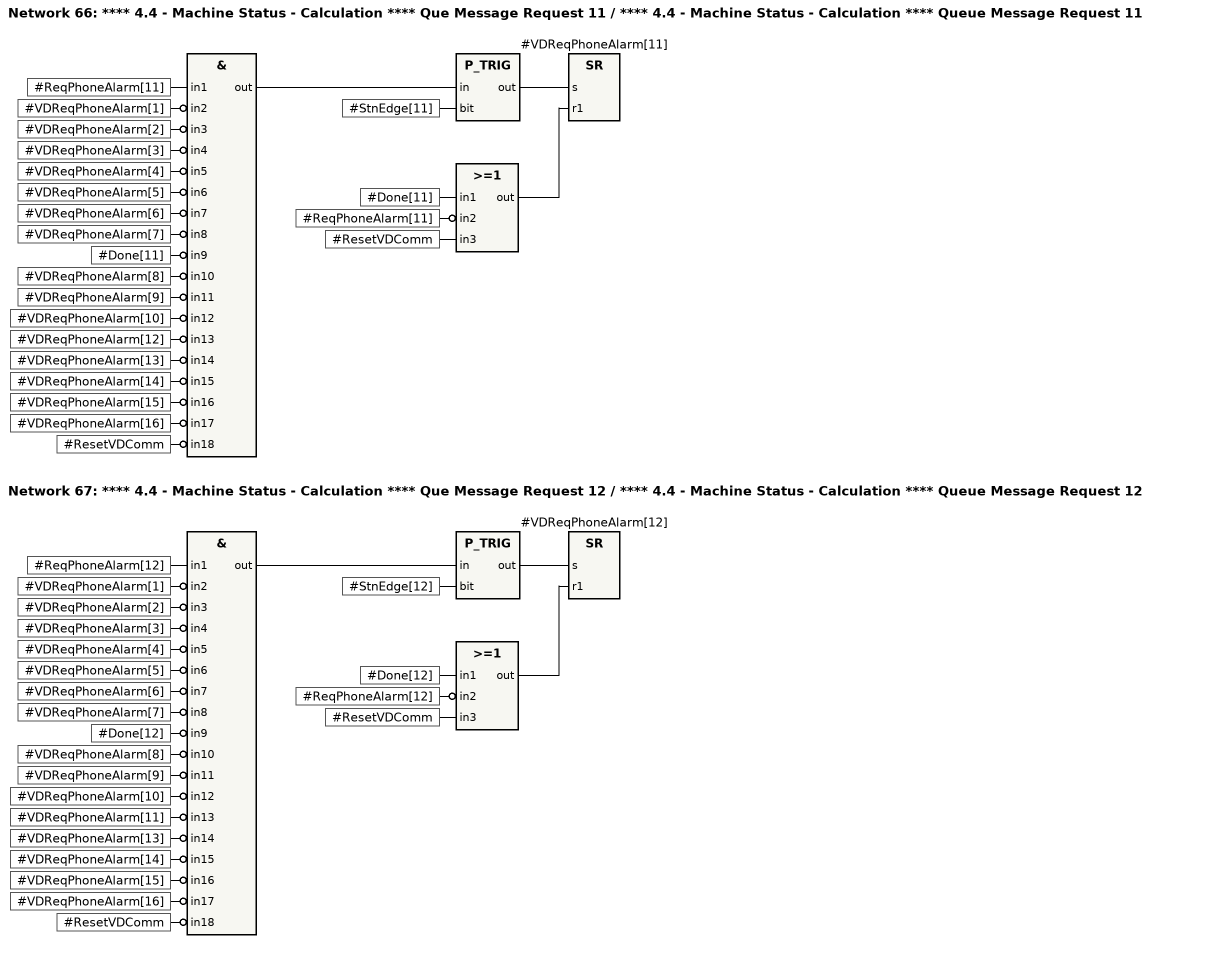
   #_w1 := #ReqPhoneAlarm[11] AND NOT #VDReqPhoneAlarm[1] AND NOT #VDReqPhoneAlarm[2] AND NOT #VDReqPhoneAlarm[3] AND NOT #VDReqPhoneAlarm[4] AND NOT #VDReqPhoneAlarm[5] AND NOT #VDReqPhoneAlarm[6] AND NOT #VDReqPhoneAlarm[7] AND NOT #Done[11] AND NOT #VDReqPhoneAlarm[8] AND NOT #VDReqPhoneAlarm[9] AND NOT #VDReqPhoneAlarm[10] AND NOT #VDReqPhoneAlarm[12] AND NOT #VDReqPhoneAlarm[13] AND NOT #VDReqPhoneAlarm[14] AND NOT #VDReqPhoneAlarm[15] AND NOT #VDReqPhoneAlarm[16] AND NOT #ResetVDComm;
   #_w2 := #_w1 AND NOT #StnEdge[11];   // rising edge
   #StnEdge[11] := #_w1;
   IF #_w2 THEN
       #VDReqPhoneAlarm[11] := TRUE;   // SR flip-flop
   END_IF;
   IF #Done[11] OR NOT #ReqPhoneAlarm[11] OR #ResetVDComm THEN #VDReqPhoneAlarm[11] := FALSE; END_IF;
END_REGION

REGION Network 67: **** 4.4 - Machine Status - Calculation **** Que Message Request 12 / **** 4.4 - Machine Status - Calculation **** Queue Message Request 12
   // Que Message Request 12 / Queue Message Request 12
   #_w1 := #ReqPhoneAlarm[12] AND NOT #VDReqPhoneAlarm[1] AND NOT #VDReqPhoneAlarm[2] AND NOT #VDReqPhoneAlarm[3] AND NOT #VDReqPhoneAlarm[4] AND NOT #VDReqPhoneAlarm[5] AND NOT #VDReqPhoneAlarm[6] AND NOT #VDReqPhoneAlarm[7] AND NOT #Done[12] AND NOT #VDReqPhoneAlarm[8] AND NOT #VDReqPhoneAlarm[9] AND NOT #VDReqPhoneAlarm[10] AND NOT #VDReqPhoneAlarm[11] AND NOT #VDReqPhoneAlarm[13] AND NOT #VDReqPhoneAlarm[14] AND NOT #VDReqPhoneAlarm[15] AND NOT #VDReqPhoneAlarm[16] AND NOT #ResetVDComm;
   #_w2 := #_w1 AND NOT #StnEdge[12];   // rising edge
   #StnEdge[12] := #_w1;
   IF #_w2 THEN
       #VDReqPhoneAlarm[12] := TRUE;   // SR flip-flop
   END_IF;
   IF #Done[12] OR NOT #ReqPhoneAlarm[12] OR #ResetVDComm THEN #VDReqPhoneAlarm[12] := FALSE; END_IF;
END_REGION

